// TwinCAT 3 PLC project TcoCore
// Title: TcoCore
// Company: Vortex.Library
// Author: Inxton
// ProjectVersion: 0.6.0.913
// ProgramVersion: 3.1.4024.12
// libraries:
//   Tc2_Standard, * (Beckhoff Automation GmbH)
//   Tc2_System, * (Beckhoff Automation GmbH)
//   Tc3_Module, * (Beckhoff Automation GmbH)
//   Tc2_EtherCAT,newest,Beckhoff Automation GmbH
//   Tc3_JsonXml,newest,Beckhoff Automation GmbH
// project tree:
//   / MAIN.TcPOU, PlcTask.TcTTO
//   POUs/Compatibility/ TcoContextCompatibility.TcPOU, TcoContextNfCompatibility.TcPOU
//   POUs/ImplicitChecks/ CheckBounds.TcPOU, CheckDivDInt.TcPOU, CheckDivLInt.TcPOU, CheckDivLReal.TcPOU, CheckDivReal.TcPOU, CheckLRangeSigned.TcPOU, CheckLRangeUnsigned.TcPOU, CheckPointer.TcPOU, CheckRangeSigned.TcPOU, CheckRangeUnsigned.TcPOU
//   POUs/Prototypes/Abstractions/ ITcoCoordinator.TcIO
//   POUs/Prototypes/TcoComponent/ ITcoComponent.TcIO, TcoComponent.TcPOU, TcoSignalInfo.TcPOU, ITcoServiceable.TcIO
//   POUs/Prototypes/TcoContext/ ITcoContextEnvironment.TcIO, TcoContextEnvironment.TcPOU, TcoContext.TcPOU, ITcoContext.TcIO
//   POUs/Prototypes/TcoDialog/TcoCustomizedDialog/ eCustomizedDialogAnswer.TcDUT, ITcoCustomizedDialogAnswer.TcIO (not stored), ITcoCustomizedDialogFormat.TcIO, TcoCustomizedDialog.TcPOU
//   POUs/Prototypes/TcoDialog/ eDialogAnswer.TcDUT, eDialogType.TcDUT, ITcoDialogAnswer.TcIO, ITcoDialogFormat.TcIO, TcoDialog.TcPOU, TcoDialogBase.TcPOU
//   POUs/Prototypes/TcoDialog/TcoInputDialog/ eInputDialogAnswer.TcDUT, ITcoInputDialogAnswer.TcIO, ITcoInputDialogFormat.TcIO, TcoInputDialog.TcPOU, TcoInputDialogContentContainer.TcPOU
//   POUs/Prototypes/TcoLogger/ ITcoLogger.TcIO, TcoLogger.TcPOU, TcoLogItem.TcDUT
//   POUs/Prototypes/TcoMessage/ eMessageCategory.TcDUT, eMessageCondition.TcDUT, eMessageDigestMethod.TcDUT, eMessengerLogMethod.TcDUT, ITcoMessageTextBuilder.TcIO, ITcoMessageProperties.TcIO, ITcoMessageCategorize.TcIO, ITcoMessenger.TcIO, ITcoMessengerEnv.TcIO, ITcoMessages.TcIO, TcoMessageDigest.TcDUT, TcoMessenger.TcPOU, TcoMessage.TcDUT, TcoMessengerEnv.TcPOU
//   POUs/Prototypes/TcoMomentaryTask/ ITcoMomentaryTask.TcIO, TcoMomentaryTask.TcPOU
//   POUs/Prototypes/TcoNothing/ NO.TcPOU
//   POUs/Prototypes/TcoObject/ ITcoObject.TcIO, TcoObject.TcPOU
//   POUs/Prototypes/TcoRemoteTask/ TcoRemoteTask.TcPOU
//   POUs/Prototypes/TcoRestorable/ ITcoObjectRestorer.TcIO, ITcoRestorable.TcIO
//   POUs/Prototypes/TcoRtc/ ITcoRtc.TcIO, RtcPrg.TcPOU, RtcSynchParams.TcDUT, TcoRtc.TcPOU
//   POUs/Prototypes/TcoSelector/ ITcoSelector.TcIO
//   POUs/Prototypes/TcoSequencer/ eStepIdUniquenessControlState.TcDUT, eSequencerMode.TcDUT, eStepStatus.TcDUT, eSequencerError.TcDUT, ITcoSequencerModeController.TcIO, TcoSequence.TcPOU, TcoSequencer.TcPOU, TcoSequencerModeController.TcPOU, TcoSequencerBase.TcPOU, ITcoSequencer.TcIO, StepDetails.TcDUT
//   POUs/Prototypes/TcoSequencer/TcoSequencerObserver/ ITcoSequencerObserver.TcIO, TcoSequencerObserver.TcPOU, TcoTcoSequencerObserverDummy.TcPOU
//   POUs/Prototypes/TcoState/ eRestoreMode.TcDUT, ITcoState.TcIO, TcoStateBase.TcPOU, TcoState.TcPOU, TcoStateExtendible.TcPOU
//   POUs/Prototypes/TcoStruct/ TcoParentedStructure.TcPOU, TcoStruct.TcDUT
//   POUs/Prototypes/TcoTask/ eTaskState.TcDUT, ITcoTaskStatus.TcIO, ITcoTask.TcIO, TcoTask.TcPOU
//   POUs/Prototypes/TcoTask/TaskResult/ TcoTaskResult.TcPOU, F_AnyToUnionValue.TcDUT
//   POUs/Prototypes/TcoTier/ TcoTier.TcPOU
//   POUs/Prototypes/TcoToggleTask/ ITcoToggleTask.TcIO, TcoToggleTask.TcPOU
//   POUs/TestFixtures/ _internals_TcoContext.TcPOU, _internals_TcoSequencer.TcPOU, _internals_TcoSequence.TcPOU
//   POUs/Utilities/ TcoCRC_16.TcPOU, TcoCRC_32.TcPOU, TcoCRC_8.TcPOU, StringBuilder.TcPOU
// real-time tasks:
//   TASK PlcTask: cycle T#10ms, priority 20, ADS port 350
//   TASK PlcTask1: cycle T#10ms, priority 21, ADS port 351
//   TASK PlcTask2: cycle T#10ms, priority 22, ADS port 352

CONFIGURATION TcoCore
    RESOURCE PLC ON TwinCAT3
        TASK PlcTask(INTERVAL := T#10ms, PRIORITY := 20);
        PROGRAM MAIN WITH PlcTask : MAIN;
    END_RESOURCE
END_CONFIGURATION

// ---- POUs/Prototypes/TcoDialog/TcoCustomizedDialog/eCustomizedDialogAnswer.TcDUT
{attribute 'qualified_only'}
{attribute 'strict'}
TYPE eCustomizedDialogAnswer :
(
    NoAnswer := 0,
    Option1 := 10,
    Option2 := 20,
    Option3 := 30,
    Option4 := 40,
    Invoked := 50
);
END_TYPE

// ---- POUs/Prototypes/TcoDialog/eDialogAnswer.TcDUT
{attribute 'qualified_only'}
{attribute 'strict'}
TYPE eDialogAnswer :
(
    NoAnswer := 0,
    OK := 10,
    Yes := 20,
    No := 30,
    Cancel := 40,
    Invoked := 50
);
END_TYPE

// ---- POUs/Prototypes/TcoDialog/eDialogType.TcDUT
{attribute 'qualified_only'}
{attribute 'strict'}
TYPE eDialogType :
(
    Undefined := 0,
    Info := 10,
    Question := 20,
    Warning := 30,
    Error := 40
);
END_TYPE

// ---- POUs/Prototypes/TcoDialog/TcoInputDialog/eInputDialogAnswer.TcDUT
{attribute 'qualified_only'}
{attribute 'strict'}
TYPE eInputDialogAnswer :
(
    NoAnswer := 0,
    OK := 10,
    Yes := 20,
    No := 30,
    Cancel := 40,
    Invoked := 50
);
END_TYPE

// ---- POUs/Prototypes/TcoLogger/TcoLogItem.TcDUT
(*~
    <docu>
        <summary>
            Logger message object contains complete message details including time stamp, message text, message category, identity of the message provider, context cycle in which the message was posted.
        </summary>
    </docu>
~*)
TYPE TcoLogItem :
STRUCT
    (*~
    <docu>
        <summary>
            Time when the message was posted.
        </summary>
    </docu>
~*)
    {attribute clr [ReadOnly()]}
    TimeStamp : DT;
    (*~
    <docu>
        <summary>
            Text of the message.
        </summary>
    </docu>
~*)
    {attribute clr [ReadOnly()]}
    Text : STRING(TcoMessengerEnv.MAX_MESSAGE_TEXT_LENGHT);
    (*~
    <docu>
        <summary>
            Identity of the TcoObject that posted this message.
        </summary>
    </docu>
~*)
    {attribute clr [ReadOnly()]}
    Identity : ULINT;
    (*~
    <docu>
        <summary>
            Message category of this message. See <see cref="TcoCore.eMessageCategory"/> for detailed informations.
        </summary>
    </docu>
~*)
    Category : eMessageCategory;
    (*~
    <docu>
        <summary>
            Context cycle in which the message was posted.
        </summary>
    </docu>
~*)
    {attribute clr [ReadOnly()]}
    Cycle : ULINT;
    (*~
    <docu>
        <summary>
            Count of messages of the object in the current cycle.
        </summary>
    </docu>
~*)
    {attribute clr [ReadOnly()]}
    PerCycleCount : BYTE;
    (*~
    <docu>
        <summary>
            Indicates that the message is expected to be dequeed from the buffer.
        </summary>
    </docu>
~*)
    ExpectDequeing : BOOL;
    (*~
    <docu>
        <summary>
            Stores message digest of this message text.
        </summary>
    </docu>
    ~*)
    MessageDigest : DWORD;
END_STRUCT
END_TYPE

// ---- POUs/Prototypes/TcoMessage/eMessageCategory.TcDUT
(*~
    <docu>
        <summary>
            Message categories.
        </summary>
    </docu>
~*)
// ATTENTION: Values must be multiply of 100
{attribute 'qualified_only'}
{attribute 'strict'}
TYPE eMessageCategory :
(
    All := 0,
    (*~
    <docu>
        <summary>
            Trace message to be used for tracing purpose.
            Use when you need to track detailed information about internal states of the program for detailed visibility.
            This is lowest level of category that can be used in production, for detailed observation of PLC program.
        </summary>
    </docu>
    ~*)
    Trace := 100,
    (*~
    <docu>
        <summary>
            Debug message to be used for debugging purpose only.
            Use when you need to report debug information for you as programmer.
        </summary>
    </docu>
    ~*)
    Debug := 200,
    (*~
    <docu>
        <summary>
            Info message.
            Use when you want to deliver information to the user, that has only informative character and does not adversely affect a process.
        </summary>
    </docu>
    ~*)
    Info := 300,
    (*~
    <docu>
        <summary>
            Time-out message.
            Use this category when you want to report a timed-out information, that may eventually succed.
        </summary>
    </docu>
    ~*)
    TimedOut := 400,
    (*~
    <docu>
        <summary>
            Notification message.
            Use this category when you want to report a notification that may be of interest to the user, but does not adversly affect a process.
        </summary>
    </docu>
    ~*)
    Notification := 500,
    (*~
    <docu>
        <summary>
            Warning message.
            Use this category when you want to report to the user an information about a possible problem, that may adversly affect a process.
            Information in this cateogory aims to help the user to identify a problem, the cause of such problem does not necessarily stops the process.
        </summary>
    </docu>
    ~*)
    Warning := 600,
    (*~
    <docu>
        <summary>
            Error message.
            Use this categoty when there is a failure that cannot be immediately recovered and an intervention is needed. This is typically a situation when a device fails
            to deliver expected result.
            Do not use this category to report information about failed process like measurement or detection.
        </summary>
    </docu>
    ~*)
    Error := 700,
    (*~
    <docu>
        <summary>
            Programming issue.
            Use this category to inform about a possible programming error, defect in settings or missing information at a level of programming or system or process settings.
        </summary>
    </docu>
    ~*)
    ProgrammingError := 900,
    (*~
    <docu>
        <summary>
            Critical error.
            Use this category when a critical error occured, that is not recoverable by the means of software (reset/restore) and but device still operates under such conditions; a detailed inspection and an expert action is required.
        </summary>
    </docu>
    ~*)
    Critical := 1000,
    (*~
    <docu>
        <summary>
            Fatal error.
            Use this category when a fatal error occured, that is not recoverable by the means of software (reset/restore) and a detailed inspection is required, the device is not able to continue without special intervention,
        </summary>
    </docu>
    ~*)
    Fatal := 1100,
    (*~
    <docu>
        <summary>
            Catastrophic error.
            Use this category when there is a situation when the device cannot continue operations due to irrecoverable failure.
        </summary>
    </docu>
    ~*)
    Catastrophic := 1200,
    None := 32000
);
END_TYPE

// ---- POUs/Prototypes/TcoMessage/eMessageCondition.TcDUT
{attribute 'qualified_only'}
{attribute 'strict'}
TYPE INTERNAL eMessageCondition :
(
    Unconditional := 0,
    Active := 10,
    Inactive := 20
);
END_TYPE

// ---- POUs/Prototypes/TcoMessage/eMessageDigestMethod.TcDUT
(*~
    <docu>
        <summary>
            Message digest methods used to create fingerprint of a message.
        </summary>
    </docu>
~*)
{attribute 'qualified_only'}
{attribute 'strict'}
TYPE eMessageDigestMethod :
(
    (*~
    <docu>
        <summary>
             Fastest method with highest probability of colisions.
        </summary>
    </docu>
    ~*)
    CRC8 := 8,
    (*~
    <docu>
        <summary>
             Moderate speed method with lower probability of colisions.
        </summary>
    </docu>
    ~*)
    CRC16 := 16,
    (*~
    <docu>
        <summary>
             Slowest speed method with relatively low probability of colisions.
        </summary>
    </docu>
    ~*)
    CRC32 := 32,
    (*~
    <docu>
        <summary>
             Messages are not digested the repeated messages won't be filtered out.
             Use this option on low performance devices.
        </summary>
    </docu>
    ~*)
    NONE := 32767
);
END_TYPE

// ---- POUs/Prototypes/TcoMessage/eMessengerLogMethod.TcDUT
(*~
    <docu>
        <summary>
            Message logging method. Determines how the messages will be pushed to the log buffer.
        </summary>
    </docu>
~*)
{attribute 'qualified_only'}
{attribute 'strict'}
TYPE eMessengerLogMethod :
(
    (*~
    <docu>
        <summary>
            Logs message when the occurence of the message content arises.
            If the message with the same content occurs in the n+1 cycle such message is not pushed.
        </summary>
    </docu>
    ~*)
    OnEventRisen := 100,
    (*~
    <docu>
        <summary>
            Logs message continuosly with not filtering.
            <note type="important">This method may easily overrun the circular message buffer.</note>
        </summary>
    </docu>
    ~*)
    Continuous := 200,
    (*~
    <docu>
        <summary>
            No logging.
        </summary>
    </docu>
    ~*)
    NoLogging := 300
);
END_TYPE

// ---- POUs/Prototypes/TcoMessage/TcoMessageDigest.TcDUT
TYPE TcoMessageDigest :
STRUCT
    Digest : DWORD;
    Cycle : ULINT;
    Count : ULINT;
    Category : eMessageCategory;
END_STRUCT
END_TYPE

// ---- POUs/Prototypes/TcoMessage/TcoMessage.TcDUT
(*~
    <docu>
        <summary>
            Complete message details including time stamp, message text, message category, identity of the message provider, context cycle in which the message was posted.
        </summary>
    </docu>
~*)
TYPE TcoMessage :
STRUCT
    (*~
    <docu>
        <summary>
            Time when the message was posted.
        </summary>
    </docu>
~*)
    {attribute clr [ReadOnly()]}
    TimeStamp : DT;
    (*~
    <docu>
        <summary>
            Text of the message.
        </summary>
    </docu>
~*)
    {attribute clr [ReadOnly()]}
    Text : STRING(TcoMessengerEnv.MAX_MESSAGE_TEXT_LENGHT);
    (*~
    <docu>
        <summary>
            Identity of the TcoObject that posted this message.
        </summary>
    </docu>
~*)
    {attribute clr [ReadOnly()]}
    Identity : ULINT;
    (*~
    <docu>
        <summary>
            Message category of this message. See <see cref="TcoCore.eMessageCategory"/> for detailed informations.
        </summary>
    </docu>
~*)
    Category : eMessageCategory;
    (*~
    <docu>
        <summary>
            Context cycle in which the message was posted.
        </summary>
    </docu>
~*)
    {attribute clr [ReadOnly()]}
    Cycle : ULINT;
    (*~
    <docu>
        <summary>
            Count of messages of the object in the current cycle.
        </summary>
    </docu>
~*)
    {attribute clr [ReadOnly()]}
    PerCycleCount : BYTE;
    (*~
    <docu>
        <summary>
            Indicates that the message is expected to be dequeed from the buffer.
        </summary>
    </docu>
~*)
    ExpectDequeing : BOOL;
    (*~
    <docu>
        <summary>
            Indicates that the message must be persisted in the alarm view until acknowledged.
        </summary>
    </docu>
    ~*)
    Pinned : BOOL;
    (*~
    <docu>
        <summary>
            Stores message digest of this message text.
        </summary>
    </docu>
    ~*)
    MessageDigest : DWORD;
END_STRUCT
END_TYPE

// ---- POUs/Prototypes/TcoRtc/RtcSynchParams.TcDUT
TYPE RtcSynchParams :
STRUCT
    synchContextIdentity : ULINT;
    doSynch : BOOL;
    syncAmsId : STRING;
    syncPeriod : UINT;
END_STRUCT
END_TYPE

// ---- POUs/Prototypes/TcoSequencer/eStepIdUniquenessControlState.TcDUT
{attribute 'qualified_only'}
{attribute 'strict'}
TYPE eStepIdUniquenessControlState :
(
    Deactivated := -1,
    NotYetStarted := 0,
    Requested := 10,
    Started := 20,
    Running := 40,
    Done := 200,
    Error := 255
);
END_TYPE

// ---- POUs/Prototypes/TcoSequencer/eSequencerMode.TcDUT
(*~
    <docu>
        <summary>
            Modes of the sequencer.
        </summary>
    </docu>
~*)
{attribute 'qualified_only'}
{attribute 'strict'}
TYPE eSequencerMode :
(
    (*~
    <docu>
        <summary>
            Invalid, no logic is executed.
        </summary>
    </docu>
~*)
    Invalid := -10,
    (*~
    <docu>
        <summary>
            Sequencer runs the steps of the sequence.
            (When cyclic mode is selected, next step is automatically started after the previous one has been completed.)
        </summary>
    </docu>
~*)
    CyclicMode := 0,
    (*~
    <docu>
        <summary>
            Sequencer is in mode of step-by-step operation. The current step completes the execution regularly.
            In this mode the Step Forward/Backward and manual step execution is available.
            <para>
                See <see cref="PlcDocu.TcoCore.TcoSequencerModeController.StepForward()"/> for detailed description.
                See <see cref="PlcDocu.TcoCore.TcoSequencerModeController.StepIn()"/> for detailed description.
                See <see cref="PlcDocu.TcoCore.TcoSequencerModeController.StepBackward()"/> for detailed description.
            </para>
        </summary>
    </docu>
~*)
    StepMode := 10
);
END_TYPE

// ---- POUs/Prototypes/TcoSequencer/eStepStatus.TcDUT
(*~
    <docu>
        <summary>
            Describes the step status inside the sequencer.
        </summary>
    </docu>
~*)
{attribute 'qualified_only'}
{attribute 'strict'}
TYPE eStepStatus :
(
    (*~
    <docu>
        <summary>
            No status defined.
        </summary>
    </docu>
~*)
    None := 0,
    (*~
    <docu>
        <summary>
            Step is disabled and won't be executed.
            Next enabled step in the sequence will be executed, when the sequencer reaches that step.
        </summary>
    </docu>
~*)
    Disabled := 10,
    (*~
    <docu>
        <summary>
            Step is ready to run. This case occurs when sequence is in step mode, step is in order of the execution and step is enabled.
            The body statements of the current step's are not executing. After calling StepIn method, step starts running the statements.
        </summary>
    </docu>
~*)
    ReadyToRun := 20,
    (*~
    <docu>
        <summary>
            Step is currently running (The body statements are running).
        </summary>
    </docu>
~*)
    Running := 30,
    (*~
    <docu>
        <summary>
            Step has finished (The body statements are not running).
        </summary>
    </docu>
~*)
    Done := 40,
    (*~
    <docu>
        <summary>
            Step is in error state. The sequencer does not execute any step logic.
        </summary>
    </docu>
~*)
    Error := 50
);
END_TYPE

// ---- POUs/Prototypes/TcoSequencer/eSequencerError.TcDUT
(*~
    <docu>
        <summary>
            Describes cause of the sequencer error.
        </summary>
    </docu>
~*)
{attribute 'qualified_only'}
{attribute 'strict'}
TYPE eSequencerError :
(
    (*~
    <docu>
        <summary>
            No error.
        </summary>
    </docu>
~*)
    noError := 0,
    (*~
    <docu>
        <summary>
            Some of the StepId in the sequence is not unique (```TcoSequencer.Step(StepID)```).
        </summary>
    </docu>
~*)
    NotUniqueStepId := 10,
    (*~
    <docu>
        <summary>
            StepId of the currently executed step has been changed during execution.
        </summary>
    </docu>
~*)
    StepIdHasBeenChanged := 20,
    (*~
    <docu>
        <summary>
            Order of the currently executed step has been changed during execution.
        </summary>
    </docu>
~*)
    OrderOfTheStepHasBeenChanged := 40,
    (*~
    <docu>
        <summary>
            Method ```RequestStep``` has been called with nonexisting StepId.
        </summary>
    </docu>
~*)
    StepWithRequestedIdDoesNotExists := 50,
    (*~
    <docu>
        <summary>
            Multiple simultaneous calls of ```RequestStep()```. Another ```RequestStep()``` method has been called while previous ```RequestStep()``` call has not yet been completed.
        </summary>
    </docu>
~*)
    MultipleRequestStepMethodCall := 60,
    (*~
    <docu>
        <summary>
            StepId is bellow min. range. Minimal value is -32767.
        </summary>
    </docu>
~*)
    StepIdTooLow := 70,
    (*~
    <docu>
        <summary>
            StepId is above max range. Maximal value is 32766.
        </summary>
    </docu>
~*)
    StepIdTooHigh := 80,
    (*~
    <docu>
        <summary>
            Mode of the sequencer is invalid.
        </summary>
    </docu>
~*)
    InvalidSequencerMode := 90
);
END_TYPE

// ---- POUs/Prototypes/TcoSequencer/StepDetails.TcDUT
(*~
    <docu>
        <summary>
            Describes the status of a step of the sequencer.
        </summary>
    </docu>
~*)
TYPE StepDetails :
STRUCT
    (*~
    <docu>
        <summary>
            Step identification number.
        </summary>
        <remarks>
             <note type="important">
                This number must be unique throughout the complete sequence. It is required to uniquely identify the step of the sequence.
            </note>
            <para>
                The <see cref="PlcDocu.TcoCore.TcoSequencer.RequestStep"/> method is using this number to jump to the required step.
            </para>
        </remarks>
    </docu>
~*)
    {attribute addProperty Name "<#Step ID#>"}
    ID : INT;
    (*~
    <docu>
        <summary>
            Order of the step in the sequence.
        </summary>
    </docu>
~*)
    {attribute addProperty Name "<#Step Order#>"}
    Order : UINT;
    (*~
    <docu>
        <summary>
            If this value is false, step body is not executed and execution is moved to the next enabled step in the sequence.
        </summary>
    </docu>
~*)
    {attribute addProperty Name "<#Enabled#>"}
    Enabled : BOOL;
    (*~
    <docu>
        <summary>
            Step description text.
        </summary>
    </docu>
~*)
    {attribute addProperty Name "<#Step description#>"}
    Description : STRING(254);
    (*~
    <docu>
        <summary>
            Describes step status.
        </summary>
        <remarks>
            <para>
                See <see cref="TcoCore.eStepStatus"/> for detailed description.
            </para>
        </remarks>
        enumStepStatus
    </docu>
~*)
    {attribute addProperty Name "<#Step status#>"}
    Status : eStepStatus;
    (*~
    <docu>
        <summary>
            Step duration time.
        </summary>
    </docu>
~*)
    {attribute addProperty Name "<#Step duration#>"}
    Duration : TIME;
END_STRUCT
END_TYPE

// ---- POUs/Prototypes/TcoState/eRestoreMode.TcDUT
{attribute 'qualified_only'}
{attribute 'strict'}
TYPE eRestoreMode :
(
    None := 0,
    (*~
    <docu>
        <summary>
                Activates automatic restore mechanism for all immediate children (direct members).
        </summary>
    </docu>
    ~*)
    AutoRestoreMembers := 10
);
END_TYPE

// ---- POUs/Prototypes/TcoStruct/TcoStruct.TcDUT
(*~
    <docu>
        <summary>
            Basic structure block from which most of the structures in TcOpen derive. `TcoStruct` provides construction mechanism to allow for access to the
            parent function block and the context.
            <note type="important">
                    The derived structure must be initialized in the declaration of the function block `mystruct : MyCustomStructure := (Parent := THIS^)`,
                    when nested in another structure `mystruct : MyCustomStructure := (Parent := THISSTRUCT)`. This will provide access to the `TcoContext`
                    and parent `TcoObject`.
            </note>
         </summary>

    </docu>
~*)
TYPE ABSTRACT TcoStruct :
STRUCT
    {attribute 'hide'}
    {attribute clr [ReadOnly()]}
    Parent : ITcoObject;
    (*~
        <docu>
            <summary>
                Provides access to parent object of this structure.
            </summary>
        </docu>
        ~*)
    {attribute 'hide'}
    {attribute clr [ReadOnly()]}
    {attribute clr [CompilerOmits("BuilderPlainer", "BuilderShadow")]}
    THISSTRUCT : TcoParentedStructure(NO.Obj, THIS^);
END_STRUCT
END_TYPE

// ---- POUs/Prototypes/TcoTask/eTaskState.TcDUT
(*~
    <docu>
        <summary>
            Describes the state of the respective task.
        </summary>
    </docu>
~*)
{attribute 'qualified_only'}
{attribute 'strict'}
TYPE eTaskState :
(
    (*~
    <docu>
        <summary>
            Task is in Ready state, the Execute() method returns FALSE.
            Task can be started by calling the Invoke() method.
        </summary>
    </docu>
~*)
    Ready := 0,
    (*~
    <docu>
        <summary>
            Task is in Requested state, if Invoke() method has been called and the Execute() method has not been called yet. The first following call of the method Execute()
            change the task state to Executing and returns TRUE, until Done or Error state is reached.
        </summary>
    </docu>
~*)
    Requested := 10,
    (*~
    <docu>
        <summary>
            When the task is in Busy state, Execute() method returns TRUE. Leaving this state is possible as follows:
            <para>1.) By calling the Abort() task gets into the Idle state.</para>
            <para>2.) By calling the DoneWhen(true) task gets into the Done state.</para>
            <para>3.) By calling the Restore() task gets into the Idle state.</para>
            <para>4.) By calling the ThrowWhen(true) task gets into the Error state.</para>
        </summary>
    </docu>
~*)
    Busy := 20,
    (*~
    <docu>
        <summary>
            Task is in Error state. To be able to start the task again the error state has to be reseted by calling the Restore() method.
        </summary>
    </docu>
~*)
    Error := 30,
    (*~
    <docu>
        <summary>
            Task is in Done state, Execute() method returns FALSE. To be able to start the task again '''rising edge''' of the calling of the Invoke() method needs to be performed.
            <p>Analogously to the xExecute signal of the <a href="https://plcopen.org/sites/default/files/downloads/creating_plcopen_compliant_function_block_libraries.pdf" title="Title"> PLCopen </a> motion function blocks.</p>
        </summary>
    </docu>
~*)
    Done := 40
);
END_TYPE

// ---- POUs/Prototypes/TcoTask/TaskResult/F_AnyToUnionValue.TcDUT
// credits Jakob Sagatowski https://github.com/sagatowski & contributors https://github.com/tcunit/TcUnit
TYPE F_AnyToUnionValue : UNION
    _bool : BOOL;
    _bit : BIT;
    _byte : BYTE;
    _dword : DWORD;
    _lword : LWORD;
    _string : STRING(255);
    _udint : UDINT;
    _uint : UINT;
    _usint : USINT;
    _sint : SINT;
    _int : INT;
    _word : WORD;
    _dint : DINT;
    _lint : LINT;
    _ulint : ULINT;
    _real : REAL;
    _lreal : LREAL;
    _wstring : WSTRING(255);
    _time : TIME;
    _ltime : LTIME;
    _date : DATE;
    _dateandtime : DATE_AND_TIME;
    _timeofday : TIME_OF_DAY;
END_UNION
END_TYPE

// ---- POUs/Prototypes/Abstractions/ITcoCoordinator.TcIO
INTERFACE ITcoCoordinator

PROPERTY IsFreshState : BOOL
GET
END_GET
END_PROPERTY

METHOD MoveNext : BOOL
END_METHOD

METHOD Retry : BOOL
VAR_INPUT
	inFromState : INT;
END_VAR
END_METHOD

METHOD Terminate : BOOL
END_METHOD

END_INTERFACE

// ---- POUs/Prototypes/TcoComponent/ITcoComponent.TcIO
INTERFACE ITcoComponent EXTENDS ITcoObject,ITcoRestorable, ITcoServiceable

END_INTERFACE

// ---- POUs/Prototypes/TcoContext/ITcoContextEnvironment.TcIO
INTERFACE ITcoContextEnvironment

PROPERTY Messaging : ITcoMessengerEnv
GET
END_GET
END_PROPERTY

END_INTERFACE

// ---- POUs/Prototypes/TcoDialog/TcoCustomizedDialog/ITcoCustomizedDialogFormat.TcIO
INTERFACE ITcoCustomizedDialogFormat

METHOD WithCaption : ITcoCustomizedDialogAnswer
VAR_INPUT
	inCaption : STRING(255);
END_VAR
END_METHOD

METHOD WithImage : ITcoCustomizedDialogAnswer
VAR_INPUT
	inSource : STRING(255);
	inHeight:REAL;
	inWidth:REAL;
END_VAR
END_METHOD

METHOD WithOption1 : ITcoCustomizedDialogAnswer
VAR_INPUT
	inContent:STRING;
END_VAR
END_METHOD

METHOD WithOption2 : ITcoCustomizedDialogAnswer
VAR_INPUT
	inContent:STRING;
END_VAR
END_METHOD

METHOD WithOption3 : ITcoCustomizedDialogAnswer
VAR_INPUT
	inContent:STRING;
END_VAR
END_METHOD

METHOD WithOption4 : ITcoCustomizedDialogAnswer
VAR_INPUT
	inContent:STRING;
END_VAR
END_METHOD

METHOD WithText : ITcoCustomizedDialogAnswer
VAR_INPUT
	inText : STRING(500);
END_VAR
END_METHOD

METHOD WithType : ITcoCustomizedDialogAnswer
VAR_INPUT
	inDialogType : eDialogType;
END_VAR
END_METHOD

END_INTERFACE

// ---- POUs/Prototypes/TcoDialog/ITcoDialogAnswer.TcIO
INTERFACE ITcoDialogAnswer EXTENDS ITcoDialogFormat

PROPERTY Answer : eDialogAnswer
GET
END_GET
END_PROPERTY

END_INTERFACE

// ---- POUs/Prototypes/TcoDialog/ITcoDialogFormat.TcIO
INTERFACE ITcoDialogFormat

METHOD WithCaption : ITcoDialogAnswer
VAR_INPUT
	inCaption : STRING(255);
END_VAR
END_METHOD

METHOD WithImage : ITcoDialogAnswer
VAR_INPUT
	inSource : STRING(255);
	inHeight:REAL;
	inWidth:REAL;
END_VAR
END_METHOD

METHOD WithOk : ITcoDialogAnswer
VAR_INPUT
END_VAR
END_METHOD

METHOD WithText : ITcoDialogAnswer
VAR_INPUT
	inText : STRING(500);
END_VAR
END_METHOD

METHOD WithType : ITcoDialogAnswer
VAR_INPUT
	inDialogType : eDialogType;
END_VAR
END_METHOD

METHOD WithYesNo : ITcoDialogAnswer
VAR_INPUT
END_VAR
END_METHOD

METHOD WithYesNoCancel : ITcoDialogAnswer
END_METHOD

END_INTERFACE

// ---- POUs/Prototypes/TcoDialog/TcoInputDialog/ITcoInputDialogAnswer.TcIO
INTERFACE ITcoInputDialogAnswer EXTENDS ITcoInputDialogFormat

PROPERTY Answer : eInputDialogAnswer
GET
END_GET
END_PROPERTY

END_INTERFACE

// ---- POUs/Prototypes/TcoDialog/TcoInputDialog/ITcoInputDialogFormat.TcIO
INTERFACE ITcoInputDialogFormat

METHOD WithCaption : ITcoInputDialogAnswer
VAR_INPUT
	inCaption : STRING(255);
END_VAR
END_METHOD

METHOD WithImage : ITcoInputDialogAnswer
VAR_INPUT
	inSource : STRING(255);
	inHeight:REAL;
	inWidth:REAL;
END_VAR
END_METHOD

METHOD WithOk : ITcoInputDialogAnswer
VAR_INPUT
END_VAR
END_METHOD

METHOD WithText : ITcoInputDialogAnswer
VAR_INPUT
	inText : STRING(500);
END_VAR
END_METHOD

METHOD WithType : ITcoInputDialogAnswer
VAR_INPUT
	inDialogType : eDialogType;
END_VAR
END_METHOD

METHOD WithYesNo : ITcoInputDialogAnswer
VAR_INPUT
END_VAR
END_METHOD

END_INTERFACE

// ---- POUs/Prototypes/TcoLogger/ITcoLogger.TcIO
INTERFACE ITcoLogger

(*~
		<docu>
			<summary>
				Pushes the message to logging buffer.
				See also `PushMessage`
				<note type="important">When using this method in a cyclical environment the message will be push each time it is called. You may easily overrun the logging buffer.</note>
			</summary>
		</docu>
~*)
METHOD PUBLIC Push
VAR_INPUT
	(*~
		<docu>
			<summary>
				Message/log entry text.
			</summary>
		</docu>
	~*)
	Text : STRING(TcoMessengerEnv.MAX_MESSAGE_TEXT_LENGHT);
	(*~
		<docu>
			<summary>
				Message/log entry category.
			</summary>
		</docu>
	~*)
	Category : eMessageCategory;
END_VAR
END_METHOD

(*~
		<docu>
			<summary>
				Pushes the message to logging buffer.
				See also `Push`
				<note:important>
						This method is typically invoked from a `TcoMessenger`.
						Depending on settings of the messenger the messages can be logged on rising edge of the message, to prevent buffer overrun.
						For details see `TcoMessengerSettings`.
				</note>
			</summary>
		</docu>
~*)
METHOD PushMessage
VAR_INPUT
	inMessage : TcoMessage;
END_VAR
END_METHOD

END_INTERFACE

// ---- POUs/Prototypes/TcoMessage/ITcoMessageTextBuilder.TcIO
INTERFACE ITcoMessageTextBuilder

METHOD Append : ITcoMessageTextBuilder
VAR_INPUT
	Text : STRING(TcoMessengerEnv.MAX_MESSAGE_TEXT_LENGHT);
END_VAR
END_METHOD

METHOD AppendAny : ITcoMessageTextBuilder
VAR_INPUT
	Data : ANY;
END_VAR
END_METHOD

METHOD As : ITcoMessageCategorize
END_METHOD

END_INTERFACE

// ---- POUs/Prototypes/TcoMessage/ITcoMessageProperties.TcIO
INTERFACE ITcoMessageProperties

METHOD Pin : ITcoMessageProperties
END_METHOD

PROPERTY Pinned : BOOL
GET
END_GET
END_PROPERTY

END_INTERFACE

// ---- POUs/Prototypes/TcoMessage/ITcoMessageCategorize.TcIO
INTERFACE ITcoMessageCategorize

(*~
		<docu>
			<summary>
				Categotizes and creates the message as 'debug'.
			</summary>
		</docu>
~*)
METHOD PUBLIC AsDebug : ITcoMessageProperties
END_METHOD

(*~
		<docu>
			<summary>
				Categotizes and creates the message as 'error'.
			</summary>
		</docu>
~*)
METHOD PUBLIC AsError : ITcoMessageProperties
END_METHOD

(*~
		<docu>
			<summary>
				Categotizes and creates the message as 'fatal'.
			</summary>
		</docu>
~*)
METHOD PUBLIC AsFatal : ITcoMessageProperties
END_METHOD

(*~
		<docu>
			<summary>
				Categotizes and creates the message as 'information'.
			</summary>
		</docu>
~*)
METHOD PUBLIC AsInfo : ITcoMessageProperties
END_METHOD

(*~
		<docu>
			<summary>
				Categotizes and creates the message as 'trace'.
			</summary>
		</docu>
~*)
METHOD PUBLIC AsTrace : ITcoMessageProperties
END_METHOD

(*~
		<docu>
			<summary>
				Categotizes and creates the message as 'warning'.
			</summary>
		</docu>
~*)
METHOD PUBLIC AsWarning : ITcoMessageProperties
END_METHOD

END_INTERFACE

// ---- POUs/Prototypes/TcoMessage/ITcoMessenger.TcIO
INTERFACE ITcoMessenger EXTENDS ITcoMessages

(*~
		<docu>
			<summary>
				Clears the message content.
				<remarks>
					<note type="important">
						This method is exposed for Rpc calls, for testing purposes. Rpc calls of this method must not be used in production code
					</note>
				</remarks>
			</summary>
		</docu>
~*)
METHOD Clear
END_METHOD

METHOD OnCondition : ITcoMessages
VAR_INPUT
	inCondition : BOOL;
END_VAR
END_METHOD

END_INTERFACE

// ---- POUs/Prototypes/TcoMessage/ITcoMessengerEnv.TcIO
INTERFACE ITcoMessengerEnv

PROPERTY IsSuspended : BOOL
GET
END_GET
END_PROPERTY

PROPERTY MessageDigestMethod : eMessageDigestMethod
GET
END_GET
SET
END_SET
END_PROPERTY

PROPERTY MessengerLoggingMethod : eMessengerLogMethod
GET
END_GET
SET
END_SET
END_PROPERTY

PROPERTY MinLevel : eMessageCategory
GET
END_GET
SET
END_SET
END_PROPERTY

METHOD Resume : BOOL
VAR_INPUT
END_VAR
END_METHOD

PROPERTY StringBuilder : REFERENCE TO StringBuilder
GET
END_GET
END_PROPERTY

METHOD Suspend
END_METHOD

END_INTERFACE

// ---- POUs/Prototypes/TcoMessage/ITcoMessages.TcIO
INTERFACE ITcoMessages

METHOD Build : ITcoMessageTextBuilder
END_METHOD

(*~
		<docu>
			<summary>
				Adds message of 'debug' category to the message queue.
			</summary>
		</docu>
~*)
METHOD PUBLIC Debug : ITcoMessageProperties
VAR_INPUT
	(*~
		<docu>
			<summary>
				Arbitrary message string.
			</summary>
		</docu>
	~*)
	Message : STRING(TcoMessengerEnv.MAX_MESSAGE_TEXT_LENGHT);
END_VAR
END_METHOD

(*~
		<docu>
			<summary>
				Adds message of 'error' category to the message queue.
			</summary>
		</docu>
~*)
METHOD PUBLIC Error : ITcoMessageProperties
VAR_INPUT
	(*~
		<docu>
			<summary>
				Arbitrary message string.
			</summary>
		</docu>
	~*)
	Message : STRING(TcoMessengerEnv.MAX_MESSAGE_TEXT_LENGHT);
END_VAR
END_METHOD

(*~
		<docu>
			<summary>
				Adds message of 'information' category to the message queue.
			</summary>
		</docu>
~*)
METHOD PUBLIC Info : ITcoMessageProperties
VAR_INPUT
	(*~
		<docu>
			<summary>
				Arbitrary message string.
			</summary>
		</docu>
	~*)
	Message : STRING(TcoMessengerEnv.MAX_MESSAGE_TEXT_LENGHT);
END_VAR
END_METHOD

(*~
		<docu>
			<summary>
				Adds message of 'notification' category to the message queue.
			</summary>
		</docu>
~*)
METHOD Notify  : ITcoMessageProperties
VAR_INPUT
	(*~
		<docu>
			<summary>
				Arbitrary message string.
			</summary>
		</docu>
	~*)
	Message : STRING(TcoMessengerEnv.MAX_MESSAGE_TEXT_LENGHT);
END_VAR
END_METHOD

(*~
		<docu>
			<summary>
				Adds message of given category to the message queue.
			</summary>
			<returns>Message index.</returns>
		</docu>
~*)
METHOD PUBLIC Post  : ITcoMessageProperties
VAR_INPUT
	(*~
		<docu>
			<summary>
				Arbitrary message string.
			</summary>
		</docu>
	~*)
	Message : STRING(TcoMessengerEnv.MAX_MESSAGE_TEXT_LENGHT);
	(*~
		<docu>
			<summary>
				Message category.
			</summary>
		</docu>
	~*)
	Category : eMessageCategory;
END_VAR
END_METHOD

(*~
		<docu>
			<summary>
				Adds message of 'programming error' category to the message queue.
			</summary>
		</docu>
~*)
METHOD PUBLIC Programming : ITcoMessageProperties
VAR_INPUT
	(*~
		<docu>
			<summary>
				Arbitrary message string.
			</summary>
		</docu>
	~*)
	Message : STRING(TcoMessengerEnv.MAX_MESSAGE_TEXT_LENGHT);
END_VAR
END_METHOD

(*~
		<docu>
			<summary>
				Adds message of 'trace' category to the message queue.
			</summary>
		</docu>
~*)
METHOD PUBLIC Trace : ITcoMessageProperties
VAR_INPUT
	(*~
		<docu>
			<summary>
				Arbitrary message string.
			</summary>
		</docu>
	~*)
	Message : STRING(TcoMessengerEnv.MAX_MESSAGE_TEXT_LENGHT);
END_VAR
END_METHOD

(*
	<docu>
		<summary>
			Unpins this messenger.
		</summary>
	</docu>
*)
METHOD UnPin
END_METHOD

(*~
		<docu>
			<summary>
				Adds message of 'warning' category to the message queue.
			</summary>
		</docu>
~*)
METHOD PUBLIC Warning : ITcoMessageProperties
VAR_INPUT
	(*~
		<docu>
			<summary>
				Arbitrary message string.
			</summary>
		</docu>
	~*)
	Message : STRING(TcoMessengerEnv.MAX_MESSAGE_TEXT_LENGHT);
END_VAR
END_METHOD

END_INTERFACE

// ---- POUs/Prototypes/TcoComponent/ITcoServiceable.TcIO
INTERFACE ITcoServiceable

PROPERTY IsService : BOOL
GET
END_GET
END_PROPERTY

METHOD PUBLIC Service
END_METHOD

END_INTERFACE

// ---- POUs/Prototypes/TcoContext/ITcoContext.TcIO
INTERFACE ITcoContext EXTENDS ITcoObject

PROPERTY EndCycleCount : ULINT
GET
END_GET
END_PROPERTY

PROPERTY Environment : ITcoContextEnvironment
GET
END_GET
END_PROPERTY

PROPERTY Logger : ITcoLogger
GET
END_GET
END_PROPERTY

PROPERTY RealTimeClock : ITcoRtc
GET
END_GET
END_PROPERTY

PROPERTY StartCycleCount : ULINT
GET
END_GET
END_PROPERTY

END_INTERFACE

// ---- POUs/Prototypes/TcoMomentaryTask/ITcoMomentaryTask.TcIO
INTERFACE ITcoMomentaryTask EXTENDS ITcoObject

(*~
	<docu>
		<summary>
			Use to set the state of the '''TcoMomentaryOnTask''' to the value '''FALSE'''.
		</summary>
	</docu>
~*)
METHOD Off : BOOL
END_METHOD

(*~
	<docu>
		<summary>
			Use to set the state of the '''TcoMomentaryOnTask''' to the value '''TRUE'''.
		</summary>
	</docu>
~*)
METHOD On : BOOL
END_METHOD

END_INTERFACE

// ---- POUs/Prototypes/TcoObject/ITcoObject.TcIO
INTERFACE ITcoObject EXTENDS __SYSTEM.IQueryInterface

{attribute 'hide'}
PROPERTY Context : ITcoContext
GET
END_GET
END_PROPERTY

PROPERTY Identity : ULINT
GET
END_GET
END_PROPERTY

END_INTERFACE

// ---- POUs/Prototypes/TcoRestorable/ITcoObjectRestorer.TcIO
INTERFACE ITcoObjectRestorer

(*~
	<docu>
		<summary>
			Ensures calling the <c>Restore()</c> method on the object entered.
			<para>
				<example>
				<note type="Example">
				<para>
					Possibility to use the fluent syntax.
				</para>
					<code>ChangeState(newState).RestoreObject(myFirstChildObject).RestoreObject(mySecondChildObject);</code>
				 </note>
				</example>
			</para>
		</summary>
	</docu>
~*)
METHOD RestoreObject : ITcoObjectRestorer
VAR_INPUT
	Obj : ITcoRestorable;
END_VAR
END_METHOD

END_INTERFACE

// ---- POUs/Prototypes/TcoRestorable/ITcoRestorable.TcIO
INTERFACE ITcoRestorable EXTENDS __SYSTEM.IQueryInterface

METHOD Restore : ITcoRestorable
END_METHOD

END_INTERFACE

// ---- POUs/Prototypes/TcoRtc/ITcoRtc.TcIO
INTERFACE ITcoRtc

PROPERTY IsSynchronized : BOOL
GET
END_GET
END_PROPERTY

PROPERTY IsValid : BOOL
GET
END_GET
END_PROPERTY

METHOD NowLocal : DATE_AND_TIME
END_METHOD

METHOD NowLocalAsTIMESTRUCT : Tc2_EtherCAT.Tc2_Utilities.TIMESTRUCT
END_METHOD

METHOD NowUTC : DATE_AND_TIME
END_METHOD

METHOD NowUTCAsTIMESTRUCT : Tc2_EtherCAT.Tc2_Utilities.TIMESTRUCT
END_METHOD

METHOD TickClock : ULINT
END_METHOD

END_INTERFACE

// ---- POUs/Prototypes/TcoSelector/ITcoSelector.TcIO
INTERFACE ITcoSelector EXTENDS ITcoState

METHOD RequestState
VAR_INPUT
	State : INT;
END_VAR
END_METHOD

END_INTERFACE

// ---- POUs/Prototypes/TcoSequencer/ITcoSequencerModeController.TcIO
INTERFACE ITcoSequencerModeController

(*~
	<docu>
		<summary>
			Gets or sets sequencer mode.
			<remarks>
				<para>
					See <see cref="TcoCore.eSequencerMode"/> for detailed description.
				</para>
			</remarks>
		</summary>
	</docu>
~*)
PROPERTY PUBLIC Mode : eSequencerMode
GET
END_GET
SET
END_SET
END_PROPERTY

(*~
	<docu>
		<summary>
			This method triggers StepBackward task, that decrements current step (variable: <c> TcoSequencer._theOrderOfTheCurrentlyExecutedStep</c> ), in case the sequencer is in step mode, and the current step is greather than zero.
		</summary>
	</docu>
~*)
METHOD PUBLIC FINAL StepBackward
END_METHOD

(*~
	<docu>
		<summary>
			This method triggers StepForward task, that increment current step (variable: <c>TcoSequencer._theOrderOfTheCurrentlyExecutedStep</c> ),
			in case the sequencer is in step mode, and the current step is lower than number of steps in th sequence (variable: <c>TcoSequencer._numberOfStepsInSequence</c> ).
		</summary>
	</docu>
~*)
METHOD PUBLIC FINAL StepForward
END_METHOD

(*~
	<docu>
		<summary>
			Triggers StepIn task, that changes the current step status from ReadyToRun to Running.
			This causes starting the execution of the body of the current step.
		</summary>
	</docu>
~*)
METHOD PUBLIC FINAL StepIn
END_METHOD

END_INTERFACE

// ---- POUs/Prototypes/TcoSequencer/TcoSequencerObserver/ITcoSequencerObserver.TcIO
INTERFACE ITcoSequencerObserver

METHOD Observe
VAR_INPUT

	(*~
	<docu>
		<summary>
			Indicates that a step is active.
		</summary>
	</docu>
	~*)

	inIsStepActive : BOOL;
	(*~
	<docu>
		<summary>
			Currently running step order.
		</summary>
	</docu>
	~*)

	inCurrentStepOrder : UINT;
	(*~
	<docu>
		<summary>
			Step identification number.
		</summary>
		<remarks>
 			<note type="important">
				This number must be unique throughout the complete sequence. It is required to uniquely identify the step of the sequence.
			</note>
			<para>
				The <see cref="PlcDocu.TcoCore.TcoSequencer.RequestStep"/> method is using this number to jump to the required step.
			</para>
		</remarks>
	</docu>
	~*)
		{attribute addProperty Name "<#Step ID#>"}
		inID: INT;
	(*~
		<docu>
			<summary>
				Order of the step in the sequence.
			</summary>
		</docu>
	~*)
		{attribute addProperty Name "<#Step Order#>"}
		inOrder: UINT;
	(*~
		<docu>
			<summary>
				If this value is false, step body is not executed and execution is moved to the next enabled step in the sequence.
			</summary>
		</docu>
	~*)
		{attribute addProperty Name "<#Enabled#>"}
		inEnabled: BOOL;
	(*~
		<docu>
			<summary>
				Step description text.
			</summary>
		</docu>
	~*)
		{attribute addProperty Name "<#Step description#>"}
		inDescription: STRING(254);
	(*~
		<docu>
			<summary>
				Describes step status.
			</summary>
			<remarks>
				<para>
					See <see cref="TcoCore.eStepStatus"/> for detailed description.
				</para>
			</remarks>
			enumStepStatus
		</docu>
	~*)
		{attribute addProperty Name "<#Step status#>"}
		inStatus : eStepStatus;
	(*~
		<docu>
			<summary>
				Step duration time.
			</summary>
		</docu>
	~*)
		{attribute addProperty Name "<#Step duration#>"}
		inDuration : TIME;

			(*~
		<docu>
			<summary>
				Total steps count;
			</summary>
		</docu>
	~*)
		{attribute addProperty Name "<#Step count#>"}
		inStepCount : UINT;
END_VAR
END_METHOD

END_INTERFACE

// ---- POUs/Prototypes/TcoSequencer/ITcoSequencer.TcIO
INTERFACE ITcoSequencer EXTENDS ITcoState

(*~
	<docu>
		<summary>
			Gets the information about the current step.
		</summary>
	</docu>
~*)
PROPERTY CurrentStep : REFERENCE TO StepDetails
GET
END_GET
END_PROPERTY

PROPERTY ModeController : ITcoSequencerModeController
GET
END_GET
END_PROPERTY

(*~
	<docu>
		<summary>
			<para>
				Ensures calling the Open(), Main() and Close() methods in the desired order.
				This method is final, so it cannot be overloaded. The InstanceName.Run() needs to be called cyclically inside the appropriate context.
			</para>
		</summary>
	</docu>
~*)
METHOD PUBLIC FINAL Run
END_METHOD

END_INTERFACE

// ---- POUs/Prototypes/TcoState/ITcoState.TcIO
INTERFACE ITcoState EXTENDS ITcoObject, ITcoRestorable

PROPERTY IsAutoRestoreEnabled : BOOL
GET
END_GET
END_PROPERTY

PROPERTY LastStateChangeCycle : ULINT
GET
END_GET
END_PROPERTY

METHOD RestoreObject : ITcoObjectRestorer
VAR_INPUT
	Obj : ITcoRestorable;
END_VAR
END_METHOD

PROPERTY State : INT
GET
END_GET
END_PROPERTY

END_INTERFACE

// ---- POUs/Prototypes/TcoTask/ITcoTaskStatus.TcIO
INTERFACE ITcoTaskStatus

PROPERTY Busy : BOOL
GET
END_GET
END_PROPERTY

PROPERTY Done : BOOL
GET
END_GET
END_PROPERTY

PROPERTY Error : BOOL
GET
END_GET
END_PROPERTY

END_INTERFACE

// ---- POUs/Prototypes/TcoTask/ITcoTask.TcIO
INTERFACE ITcoTask EXTENDS ITcoObject, ITcoRestorable

METHOD Abort
END_METHOD

PROPERTY Busy : BOOL
GET
END_GET
END_PROPERTY

PROPERTY Done : BOOL
GET
END_GET
END_PROPERTY

PROPERTY Error : BOOL
GET
END_GET
END_PROPERTY

(*~
	<docu>
		<summary>
			Use to start the execution of the task. The starting is possible from Ready state.
			<para>Moreover it is also possible to start the task again from Done state by performing the '''rising edge''' of the calling of the Invoke() method.</para>
			<p>Analogously to the xExecute signal of the <a href="https://plcopen.org/sites/default/files/downloads/creating_plcopen_compliant_function_block_libraries.pdf" title="Title"> PLCopen </a> motion function blocks.</p>
		</summary>
	</docu>
~*)
METHOD Invoke : ITcoTaskStatus
END_METHOD

END_INTERFACE

// ---- POUs/Prototypes/TcoToggleTask/ITcoToggleTask.TcIO
INTERFACE ITcoToggleTask EXTENDS ITcoObject

(*~
	<docu>
		<summary>
			Use to set the state of the '''TcoToggleTask''' to the value '''FALSE'''.
		</summary>
	</docu>
~*)
METHOD Off : BOOL
END_METHOD

(*~
	<docu>
		<summary>
			Use to set the state of the '''TcoToggleTask''' to the value '''TRUE'''.
		</summary>
	</docu>
~*)
METHOD On : BOOL
END_METHOD

(*~
	<docu>
		<summary>
			Use to toggle the state of the '''TcoToggleTask'''.
		</summary>
	</docu>
~*)
METHOD Toggle : BOOL
END_METHOD

END_INTERFACE

// ---- MAIN.TcPOU
PROGRAM INTERNAL MAIN
VAR
END_VAR

END_PROGRAM

// ---- POUs/Compatibility/TcoContextCompatibility.TcPOU
{attribute 'hide'}
{attribute clr [ExcludeFromApiDocumentation()]}
FUNCTION_BLOCK ABSTRACT TcoContextCompatibility EXTENDS TcoContext

{attribute 'hide'}
METHOD PROTECTED FINAL _Close
THIS^.Close();
END_METHOD

{attribute 'hide'}
METHOD PROTECTED FINAL _Open
THIS^.Open();
END_METHOD

END_FUNCTION_BLOCK

// ---- POUs/Prototypes/TcoContext/TcoContext.TcPOU
(*~
    <docu>
        <summary>
            Root construction container, provides context information for <c>TcoObjects</c> declared within its scope.
            This function block is ```abstract``` and cannot be instantiated.
            Use <see cref="PlcDocu.TcoCore.TcoContext.Run()"/> to run this context, ```Run``` method must be called only once per PLC Task cycle.
            Several 'TcoContext' instances can be declared and called inside one TwinCAT PlcTask, but only once per PLC cycle.
            The instance should not be accessed from several Twincat PlcTasks.
            Default implemenation of the 'TcoContext' allows its child members access properties <see cref="PlcDocu.TcoCore.TcoContext.StartCycleCount()"/>
            and <see cref="PlcDocu.TcoCore.TcoContext.EndCycleCount()"/>, messenger settings, rtc and other information related to the context of the running logic.
            <note type="tip">
                 A <c>TcoContext</c> can contain objects, components and PLC logic of one independent station of the machine,
                 while the another one can cover the same for another station.
            </note>
            <remarks>
                <note type="tip">
                    TwinCAT PlcTask and <see cref="PlcDocu.TcoCore.TcoTask()"/> refer to two different concepts.
                </note>
            </remarks>
        </summary>
        <example>
            Declaration part of the 'TcoContext' example.
        </example>
        <example>
                [!code-pas[Main](~/../TcOpen/src/TcoApplicationExamples/XaeAppExamples/PlcAppExamples/POUs/Context/VitoCorleone_Context.TcPOU?name=ContextExampleDeclarations)]
        </example>
        <example>
            Implementation part of the 'TcoContext' example.
        </example>
        <example>
                [!code-pas[Main](~/../TcOpen/src/TcoApplicationExamples/XaeAppExamples/PlcAppExamples/POUs/Context/VitoCorleone_Context.TcPOU?name=ContextExampleCode)]
        </example>
    </docu>
~*)
FUNCTION_BLOCK PUBLIC ABSTRACT TcoContext IMPLEMENTS ITcoContext
VAR
    (*~
        <docu>
            <summary>
                Identity of this <c>TcoContext</c>.
                This variable is used in the higher level applications,
                it allows to identify the context in SCADA like applications.
            </summary>
        </docu>
    ~*)
    {attribute clr [RenderIgnore()]}
    {attribute clr [ReadOnly()]}
    _Identity : ULINT;
    {attribute clr [ReadOnly()]}
    _startCycleCount : ULINT;
    {attribute clr [ReadOnly()]}
    _endCycleCount : ULINT;
    _messagingLevel : eMessageCategory;
    {attribute clr [ReadOnly()]}
    _rtc : TcoRtc;
    {attribute clr [RenderIgnore()]}
    _settings : TcoContextEnvironment;
    {attribute clr [RenderIgnore()]}
    _logger : TcoLogger(THIS^);
    _timeSychnMessenger : TcoMessenger(THIS^);
END_VAR

(*~
    <docu>
        <summary>
            This method is called implicitly at the entry point of this context (<see cref="PlcDocu.TcoCore.TcoContext.Run()"/>).
            <remarks>
                <note type="important">
                    Do not call this method explicitly!
                </note>
            </remarks>
        </summary>
    </docu>
~*)
METHOD INTERNAL FINAL Close
_endCycleCount := _startCycleCount;
END_METHOD

(*~
    <docu>
        <summary>
            Returns reference to this instance of the <see cref="PlcDocu.TcoCore.TcoContext()"/>.
        </summary>
    </docu>
~*)
PROPERTY Context : ITcoContext
GET
Context := THIS^;
END_GET
END_PROPERTY

(*~
    <docu>
        <summary>
            Gets the value of the counter incrememented by '1' at the end of each execution of this <see cref="PlcDocu.TcoCore.TcoContext()"/>.
        </summary>
    </docu>
~*)
PROPERTY EndCycleCount : ULINT
GET
EndCycleCount := _endCycleCount;
END_GET
END_PROPERTY

PROPERTY Environment : ITcoContextEnvironment
GET
Environment := _settings;
END_GET
END_PROPERTY

{attribute 'hide'}
METHOD FB_init : BOOL
VAR_INPUT
    bInitRetains : BOOL; // if TRUE, the retain variables are initialized (warm start / cold start)
    bInCopyCode : BOOL; // if TRUE, the instance afterwards gets moved into the copy code (online change)
END_VAR
_Identity := ADR(THIS^);
END_METHOD

(*~
    <docu>
        <summary>
            Returns the identity of this <see cref ="PlcDocu.TcoCore.TcoContext()"/>.
            This value is assigned when instantiated and cannot be changed at runtime.
            This member is used in the higher level applications.
        </summary>
    </docu>
~*)
PROPERTY Identity : ULINT
GET
Identity := _Identity;
END_GET
END_PROPERTY

(*~
        <docu>
            <summary>
                Gets logger for this context.
            </summary>
        </docu>
~*)
PROPERTY PUBLIC Logger : ITcoLogger
GET
Logger := _logger;
END_GET
END_PROPERTY

(*~
    <docu>
        <summary>
            Main method of the TcoContext. This is the entry point of any control logic that belongs to this context.
            The call of this method is ensured by calling the <c>InstanceName.Run()</c> method, and it must not be called explicitly.
            This method is abstract, and it must be overridden in derived block.
        </summary>
    </docu>
~*)
METHOD PROTECTED ABSTRACT Main
END_METHOD

(*~
    <docu>
        <summary>
            Called on entry into context. When overridden in derived class allows to execute an arbitrary logic prior to opening the context cycle.
            <remarks>
                <note type="important">
                    The method executes prior to opening the context. The context might not be properly initialized on first call.
                    Any information contained in the context at this point are from the last execution.
                </note>
            </remarks>
        </summary>
    </docu>
~*)
METHOD PROTECTED OnEntry
END_METHOD

(*~
    <docu>
        <summary>
            Called upon exit from the context. When overridden in derived class allows to execute an arbitrary logic after closing the context cycle.
        </summary>
    </docu>
~*)
METHOD PROTECTED OnExit
END_METHOD

(*~
    <docu>
        <summary>
            This method is called implicitly at the entry point of this context (<see cref="PlcDocu.TcoCore.TcoContext.Run()"/>).
            <remarks>
                <note type="important">
                    Do not call this method explicitly.
                </note>
            </remarks>
        </summary>
    </docu>
~*)
METHOD INTERNAL FINAL Open
_startCycleCount := _startCycleCount + 1;
_rtc.UpdateInternal();
END_METHOD

PROPERTY RealTimeClock : ITcoRtc
GET
RealTimeClock := _rtc;
END_GET
END_PROPERTY

(*~
    <docu>
        <summary>
            Syncronizes the Real Time Clock (RTC) from given source.
            <remarks>
                <note type="important">
                    There is single RTC source for entire application. All context share the same RTC source.
                </note>
            </remarks>
        </summary>
    </docu>
~*)
METHOD RtcSynchronize : REFERENCE TO TcoContext
VAR_INPUT
    (*~
        <docu>
            <summary>
                When called with true the synchronization mechanism executes.
            </summary>
        </docu>
    ~*)
    inDoSynch : BOOL;
    (*~
        <docu>
            <summary>
                ```AMS ID``` of the system against which RTC of this application will synchronize.
            </summary>
        </docu>
    ~*)
    inSyncAmsId : STRING;
    (*~
        <docu>
            <summary>
                Set the synchronisation period.
            </summary>
        </docu>
    ~*)
    inSyncPeriod : UINT;
END_VAR
VAR
    _RtcSynchParams : RtcSynchParams;
END_VAR
_RtcSynchParams.doSynch := inDoSynch;
_RtcSynchParams.syncAmsId := inSyncAmsId;
_RtcSynchParams.syncPeriod := inSyncPeriod;
_RtcSynchParams.synchContextIdentity := THIS^._Identity;
{warning disable C0357}
RtcPrg.Synchronize(_RtcSynchParams);
{warning enable C0357}
RtcSynchronize REF= THIS^;
_timeSychnMessenger.OnCondition(NOT THIS^.RealTimeClock.IsValid).Error('<#Real time clock is invalid!#>').Pin();

_timeSychnMessenger
    .OnCondition(THIS^.RealTimeClock.IsValid AND NOT THIS^.RealTimeClock.IsSynchronized).Warning('<#Real time clock is not sychronized.#>');
END_METHOD

(*~
    <docu>
        <summary>
            <para>
                This method executes of this context. It provided correct order of execution order of inner methods. Any logic of this context must be called within <see cref="PlcDocu.TcoCore.TcoContext.Main()"/>
                method. This method is final, so it cannot be overriden. The <c>InstanceName.Run()</c> needs to be called cyclically.
            </para>
        </summary>
    </docu>
~*)
METHOD PUBLIC FINAL Run
THIS^.OnEntry();
THIS^.Open();
THIS^.Main();
THIS^.Close();
THIS^.OnExit();
END_METHOD

(*~
    <docu>
        <summary>
            Gets number of executions of this context. Value of this property is incremented by '1' at the beginning of the <see cref="PlcDocu.TcoCore.TcoContext()"/>.
        </summary>
    </docu>
~*)
PROPERTY StartCycleCount : ULINT
GET
StartCycleCount := _startCycleCount;
END_GET
END_PROPERTY

END_FUNCTION_BLOCK

// ---- POUs/Prototypes/TcoRtc/TcoRtc.TcPOU
FUNCTION_BLOCK PUBLIC TcoRtc IMPLEMENTS ITcoRtc
VAR
    {attribute 'hide'}
    _isValid : BOOL := FALSE;
    {attribute 'hide'}
    _state : UINT;
    {attribute 'hide'}
    _TimeZoneID : Tc2_EtherCAT.Tc2_Utilities.E_TimeZoneID;
    {attribute 'hide'}
    _NT_GetLocalTime : Tc2_EtherCAT.Tc2_Utilities.NT_GetTime;
    {attribute 'hide'}
    _FB_TzSpecificLocalTimeToSystemTime : Tc2_EtherCAT.Tc2_Utilities.FB_TzSpecificLocalTimeToSystemTime;
    {attribute 'hide'}
    _RTC_EX2 : Tc2_EtherCAT.Tc2_Utilities.RTC_EX2;
    {attribute 'hide'}
    _PDT : Tc2_EtherCAT.Tc2_Utilities.TIMESTRUCT;
    {attribute 'hide'}
    _LocalTime : Tc2_EtherCAT.Tc2_Utilities.TIMESTRUCT;
    {attribute clr [ReadOnly()]}
    _LocalTimeDT : DATE_AND_TIME;
    {attribute 'hide'}
    _UTCTime : Tc2_EtherCAT.Tc2_Utilities.TIMESTRUCT;
    {attribute clr [ReadOnly()]}
    _UTCTimeDT : DATE_AND_TIME;
END_VAR

PROPERTY IsSynchronized : BOOL
GET
IsSynchronized := RtcPrg._isSynchronized;
END_GET
END_PROPERTY

PROPERTY IsValid : BOOL
GET
IsValid := _isValid;
END_GET
END_PROPERTY

METHOD NowLocal : DATE_AND_TIME
IF _isValid THEN
    NowLocal := _LocalTimeDT;
END_IF
END_METHOD

METHOD NowLocalAsTIMESTRUCT : Tc2_EtherCAT.Tc2_Utilities.TIMESTRUCT
IF _isValid THEN
    NowLocalAsTIMESTRUCT := _LocalTime;
END_IF
END_METHOD

METHOD NowUTC : DATE_AND_TIME
IF _isValid THEN
    NowUTC := _UTCTimeDT;
END_IF
END_METHOD

METHOD NowUTCAsTIMESTRUCT : Tc2_EtherCAT.Tc2_Utilities.TIMESTRUCT
IF _isValid THEN
    NowUTCAsTIMESTRUCT := _UTCTime;
END_IF
END_METHOD

METHOD TickClock : ULINT
TickClock := Tc2_EtherCAT.F_GetActualDcTime64();
END_METHOD

METHOD PROTECTED Update
VAR
    _diffToLastSyncInSeconds : LINT;
END_VAR
IF _state = 0 THEN
    //	_isValid := FALSE;
    _NT_GetLocalTime(NETID := '127.0.0.1.1.1', START := TRUE);

    IF _NT_GetLocalTime.BUSY AND NOT _NT_GetLocalTime.ERR THEN
        _state := _state + 10;
    END_IF
END_IF

IF _state = 10 THEN
    _NT_GetLocalTime(START := FALSE);

    IF NOT _NT_GetLocalTime.BUSY AND NOT _NT_GetLocalTime.ERR THEN
        _state := _state + 10;
    END_IF
END_IF

IF _state = 20 THEN
    _NT_GetLocalTime(START := FALSE);
    _PDT := _NT_GetLocalTime.TIMESTR;
    _isValid := TRUE;
END_IF

_RTC_EX2(EN := _isValid, PDT := _PDT);

_diffToLastSyncInSeconds := ABS(ULINT_TO_LINT(Tc2_EtherCAT.SYSTEMTIME_TO_DCTIME64(_RTC_EX2.CDT, 0, 0) -
            Tc2_EtherCAT.SYSTEMTIME_TO_DCTIME64(RtcPrg._LastSyncTimeStampInLocalTime, 0, 0))) /
    1000000000;

IF _state >= 20 AND RtcPrg._RtcSynchParams.doSynch AND _diffToLastSyncInSeconds >= RtcPrg._RtcSynchParams.syncPeriod THEN
    _state := 0;
END_IF

_LocalTime := _RTC_EX2.CDT;
_LocalTimeDT := Tc2_EtherCAT.Tc2_Utilities.SYSTEMTIME_TO_DT(_LocalTime);

IF RtcPrg._isSynchronized THEN
    _FB_TzSpecificLocalTimeToSystemTime(in := _LocalTime,
        tzInfo := RtcPrg._TimeZoneInformation,
        out => _UTCTime,
        eTzID => _TimeZoneID);

    _UTCTimeDT := Tc2_EtherCAT.Tc2_Utilities.SYSTEMTIME_TO_DT(_UTCTime);
END_IF
END_METHOD

METHOD INTERNAL UpdateInternal
THIS^.Update();
END_METHOD

END_FUNCTION_BLOCK

// ---- POUs/Prototypes/TcoRtc/RtcPrg.TcPOU
{attribute 'obsolete' := 'Should not be accessed from outside TcoCore library. Publicly accesible due to compatibility reasons.'}
PROGRAM PUBLIC RtcPrg
VAR
    {attribute 'hide'}
    _RtcSynchParams : RtcSynchParams;
    {attribute 'hide'}
    _isSynchronized : BOOL := FALSE;
    {attribute 'hide'}
    _state : UINT;
    {attribute 'hide'}
    _syncAmsIdIsLocale : BOOL;
    {attribute 'hide'}
    _FB_GetLocalAmsNetId : Tc2_EtherCAT.Tc2_Utilities.FB_GetLocalAmsNetId;
    {attribute 'hide'}
    _FB_GetTimeZoneInformation : Tc2_EtherCAT.Tc2_Utilities.FB_GetTimeZoneInformation;
    {attribute 'hide'}
    _FB_SetTimeZoneInformation : Tc2_EtherCAT.Tc2_Utilities.FB_SetTimeZoneInformation;
    {attribute 'hide'}
    _TimeZoneInformation : Tc2_EtherCAT.Tc2_Utilities.ST_TimeZoneInformation;
    {attribute 'hide'}
    _TimeZoneID : Tc2_EtherCAT.Tc2_Utilities.E_TimeZoneID;
    {attribute 'hide'}
    _startTime : Tc2_EtherCAT.T_DCTIME64;
    {attribute 'hide'}
    _endTime : Tc2_EtherCAT.T_DCTIME64;
    {attribute 'hide'}
    _getOffset : Tc2_EtherCAT.T_DCTIME64;
    {attribute 'hide'}
    _setOffset : Tc2_EtherCAT.T_DCTIME64;
    {attribute 'hide'}
    _NT_GetSyncTime : Tc2_EtherCAT.Tc2_Utilities.NT_GetTime;
    {attribute 'hide'}
    _NT_SetLocalTime : Tc2_EtherCAT.Tc2_Utilities.NT_SetLocalTime;
    {attribute 'hide'}
    _NT_GetLocalTime : Tc2_EtherCAT.Tc2_Utilities.NT_GetTime;
    {attribute 'hide'}
    _FB_TzSpecificLocalTimeToSystemTime : Tc2_EtherCAT.Tc2_Utilities.FB_TzSpecificLocalTimeToSystemTime;
    {attribute 'hide'}
    _remote2localDiff : Tc2_EtherCAT.T_DCTIME64;
    {attribute 'hide'}
    _local2SyncDiff_nanoseconds : LINT;
    {attribute 'hide'}
    _offset : ULINT;
    {attribute 'hide'}
    _syncCounter : ULINT;
    {attribute 'hide'}
    _lastSyncTick : Tc2_EtherCAT.T_DCTIME64;
    {attribute 'hide'}
    _timeTick : Tc2_EtherCAT.T_DCTIME64;
    {attribute 'hide'}
    _LocalTime : Tc2_EtherCAT.Tc2_Utilities.TIMESTRUCT;
    {attribute 'hide'}
    _UTCTime : Tc2_EtherCAT.Tc2_Utilities.TIMESTRUCT;
    {attribute 'hide'}
    _syncStartLocalTime : Tc2_EtherCAT.Tc2_Utilities.TIMESTRUCT;
    {attribute 'hide'}
    _LastSyncTimeStampInLocalTime : Tc2_EtherCAT.Tc2_Utilities.TIMESTRUCT;
    {attribute 'hide'}
    _LastSyncDiff_seconds : LINT;
END_VAR

{attribute 'obsolete' := 'MUST NOT BE CALLED EXPLICITELY!!! Use TcoCore.TcoContext.RtcSynchronize() instead!!!'}
METHOD PUBLIC Synchronize
VAR_INPUT
    inRtcSynchParams : RtcSynchParams;
END_VAR
//If there is no synchronization context identity already set, the value of this identity is used.
//So first TcoContext that calls this method set the synchronization parameters.
IF _RtcSynchParams.synchContextIdentity = 0 AND inRtcSynchParams.synchContextIdentity <> 0 THEN
    _RtcSynchParams.synchContextIdentity := inRtcSynchParams.synchContextIdentity;
END_IF

//In case that another TcoContest calls this method, it is ignored as only one could set the synchronization parameters.
IF _RtcSynchParams.synchContextIdentity <> 0 AND _RtcSynchParams.synchContextIdentity = inRtcSynchParams.synchContextIdentity THEN
    _RtcSynchParams.doSynch := inRtcSynchParams.doSynch;
    _RtcSynchParams.syncAmsId := inRtcSynchParams.syncAmsId;
    _RtcSynchParams.syncPeriod := inRtcSynchParams.syncPeriod;

    IF _NT_GetLocalTime.ERR THEN
        _NT_GetLocalTime(START := FALSE);
        _isSynchronized := FALSE;
        RETURN;
    END_IF

    IF _state = 0 THEN
        IF _RtcSynchParams.doSynch THEN
            _isSynchronized := FALSE;
            _state := _state + 10;
        ELSE
            _isSynchronized := FALSE;
            _state := 210;
        END_IF
    END_IF

    IF _state = 10 THEN
        _syncStartLocalTime := _NT_GetLocalTime.TIMESTR;
        _FB_GetLocalAmsNetId(bExecute := TRUE);

        IF _FB_GetLocalAmsNetId.bBusy AND NOT _FB_GetLocalAmsNetId.bError THEN
            _state := _state + 10;
        END_IF
    END_IF

    IF _state = 20 THEN
        _FB_GetLocalAmsNetId(bExecute := FALSE);

        IF NOT _FB_GetLocalAmsNetId.bBusy AND NOT _FB_GetLocalAmsNetId.bError THEN
            _state := _state + 10;
        END_IF
    END_IF

    IF _state = 30 THEN
        _syncAmsIdIsLocale := _RtcSynchParams.syncAmsId = _FB_GetLocalAmsNetId.AddrString OR
            _RtcSynchParams.syncAmsId = '127.0.0.1.1.1' OR
            _RtcSynchParams.syncAmsId = '';

        _state := _state + 10;
    END_IF

    IF _state = 40 THEN
        _startTime := Tc2_EtherCAT.F_GetActualDcTime64();
        _state := _state + 10;
    END_IF

    IF _state = 50 THEN
        _FB_GetTimeZoneInformation(sNetID := _RtcSynchParams.syncAmsId, bExecute := TRUE);

        IF _FB_GetTimeZoneInformation.bBusy AND NOT _FB_GetTimeZoneInformation.bError THEN
            _state := _state + 10;
        END_IF
    END_IF

    IF _state = 60 THEN
        _FB_GetTimeZoneInformation(bExecute := FALSE);

        IF NOT _FB_GetTimeZoneInformation.bBusy AND NOT _FB_GetTimeZoneInformation.bError THEN
            _state := _state + 10;
        END_IF
    END_IF

    IF _state = 70 THEN
        _TimeZoneInformation := _FB_GetTimeZoneInformation.tzInfo;
        _TimeZoneID := _FB_GetTimeZoneInformation.tzID;
        _endTime := Tc2_EtherCAT.F_GetActualDcTime64();
        _getOffset := (_endTime - _startTime) / 2;
        _state := _state + 10;
    END_IF

    IF _state = 80 THEN
        IF _syncAmsIdIsLocale THEN
            _state := 180;
        ELSE
            _state := _state + 10;
        END_IF
    END_IF

    IF _state = 90 THEN
        _startTime := Tc2_EtherCAT.F_GetActualDcTime64();
        _state := _state + 10;
    END_IF

    IF _state = 100 THEN
        _FB_SetTimeZoneInformation(sNetID := '127.0.0.1.1.1', tzInfo := _TimeZoneInformation, bExecute := TRUE);

        IF _FB_SetTimeZoneInformation.bBusy AND NOT _FB_SetTimeZoneInformation.bError THEN
            _state := _state + 10;
        END_IF
    END_IF

    IF _state = 110 THEN
        _FB_SetTimeZoneInformation(bExecute := FALSE);

        IF NOT _FB_SetTimeZoneInformation.bBusy AND NOT _FB_SetTimeZoneInformation.bError THEN
            _state := _state + 10;
        END_IF
    END_IF

    IF _state = 120 THEN
        _endTime := Tc2_EtherCAT.F_GetActualDcTime64();
        _setOffset := (_endTime - _startTime) / 2;
        _state := _state + 10;
    END_IF

    IF _state = 130 THEN
        _NT_GetSyncTime(NETID := _RtcSynchParams.syncAmsId, START := TRUE);

        IF _NT_GetSyncTime.BUSY AND NOT _NT_GetSyncTime.ERR THEN
            _state := _state + 10;
        END_IF
    END_IF

    IF _state = 140 THEN
        _NT_GetSyncTime(START := FALSE);

        IF NOT _NT_GetSyncTime.BUSY AND NOT _NT_GetSyncTime.ERR THEN
            _state := _state + 10;
        END_IF
    END_IF

    IF _state = 150 THEN
        _NT_GetSyncTime(START := FALSE);
        _offset := LREAL_TO_ULINT(ULINT_TO_LREAL(_getOffset + _setOffset) / 1000000) * 1000000;
        _offset := _offset + Tc2_EtherCAT.SYSTEMTIME_TO_DCTIME64(_NT_GetSyncTime.TIMESTR, 0, 0) + _getOffset + _setOffset;
        _LocalTime := Tc2_EtherCAT.DCTIME64_TO_SYSTEMTIME(_offset);
        _state := _state + 10;
    END_IF

    IF _state = 160 THEN
        _NT_GetSyncTime(START := FALSE);
        _NT_SetLocalTime(NETID := '127.0.0.1.1.1', TIMESTR := _LocalTime, START := TRUE);

        IF _NT_SetLocalTime.BUSY AND NOT _NT_SetLocalTime.ERR THEN
            _state := _state + 10;
        END_IF
    END_IF

    IF _state = 170 THEN
        _NT_GetSyncTime(START := FALSE);
        _NT_SetLocalTime(START := FALSE);

        IF NOT _NT_SetLocalTime.BUSY AND NOT _NT_SetLocalTime.ERR THEN
            _state := _state + 10;
        END_IF
    END_IF

    IF _state = 180 THEN
        _NT_GetSyncTime(NETID := _RtcSynchParams.syncAmsId, START := TRUE);
        _NT_GetLocalTime(NETID := '127.0.0.1.1.1', START := TRUE);

        IF _NT_GetSyncTime.BUSY AND NOT _NT_GetSyncTime.ERR AND NOT _NT_GetLocalTime.ERR THEN
            _state := _state + 10;
        END_IF
    END_IF

    IF _state = 190 THEN
        _NT_GetSyncTime(START := FALSE);
        _NT_GetLocalTime(START := FALSE);

        IF NOT _NT_GetSyncTime.BUSY AND NOT _NT_GetSyncTime.ERR AND NOT _NT_GetLocalTime.BUSY AND NOT _NT_GetLocalTime.ERR THEN
            _state := _state + 10;
        END_IF
    END_IF

    IF _state = 200 THEN
        _LastSyncTimeStampInLocalTime := _NT_GetLocalTime.TIMESTR;

        _LastSyncDiff_seconds := ULINT_TO_LINT(Tc2_EtherCAT.SYSTEMTIME_TO_DCTIME64(_LastSyncTimeStampInLocalTime, 0, 0) -
                Tc2_EtherCAT.SYSTEMTIME_TO_DCTIME64(_syncStartLocalTime, 0, 0)) /
            1000000000;

        _local2SyncDiff_nanoseconds := ULINT_TO_LINT(Tc2_EtherCAT.SYSTEMTIME_TO_DCTIME64(_NT_GetLocalTime.TIMESTR, 0, 0) -
                Tc2_EtherCAT.SYSTEMTIME_TO_DCTIME64(_NT_GetSyncTime.TIMESTR, 0, 0));

        _NT_GetSyncTime(START := FALSE);
        _NT_GetLocalTime(START := FALSE);
        _NT_SetLocalTime(START := FALSE);
        _LocalTime := _NT_GetLocalTime.TIMESTR;

        _FB_TzSpecificLocalTimeToSystemTime(in := _LocalTime,
            tzInfo := _TimeZoneInformation,
            out => _UTCTime,
            eTzID => _TimeZoneID);

        _lastSyncTick := Tc2_EtherCAT.F_GetActualDcTime64();
        _syncCounter := _syncCounter + 1;
        _state := _state + 10;
    END_IF

    IF _state = 210 THEN
        _NT_GetLocalTime(NETID := '127.0.0.1.1.1', START := TRUE);

        IF _NT_GetLocalTime.BUSY AND NOT _NT_GetLocalTime.ERR THEN
            _state := _state + 10;
        END_IF
    END_IF

    IF _state = 220 THEN
        _NT_GetLocalTime(START := FALSE);

        IF NOT _NT_GetLocalTime.BUSY AND NOT _NT_GetLocalTime.ERR THEN
            _state := _state + 10;
        END_IF
    END_IF

    IF _state = 230 THEN
        _isSynchronized := TRUE;
        _NT_GetSyncTime(START := FALSE);
        _NT_GetLocalTime(START := FALSE);
        _NT_SetLocalTime(START := FALSE);
        _timeTick := Tc2_EtherCAT.F_GetActualDcTime64();

        IF _RtcSynchParams.doSynch THEN
            IF (_timeTick - _lastSyncTick) / 1000000000 >= _RtcSynchParams.syncPeriod THEN //Ticks are in nanoseconds, sync period is in seconds
                _state := 0;
            ELSE
                _state := 210;
            END_IF
        ELSE
            _state := 210;
        END_IF
    END_IF
END_IF
END_METHOD

END_PROGRAM

// ---- POUs/Prototypes/TcoContext/TcoContextEnvironment.TcPOU
FUNCTION_BLOCK TcoContextEnvironment IMPLEMENTS ITcoContextEnvironment
VAR
    {attribute clr [RenderIgnore()]}
    _messenger : TcoMessengerEnv;
END_VAR

(*~
        <docu>
            <summary>
                Gets messaging settings of this context.
            </summary>
        </docu>
~*)
PROPERTY Messaging : ITcoMessengerEnv
GET
Messaging := _messenger;
END_GET
END_PROPERTY

END_FUNCTION_BLOCK

// ---- POUs/Prototypes/TcoMessage/TcoMessengerEnv.TcPOU
FUNCTION_BLOCK PUBLIC TcoMessengerEnv IMPLEMENTS ITcoMessengerEnv
VAR
    _minLevel : eMessageCategory;
    _isMessagingSuspended : BOOL;
    _messageDigestMethod : eMessageDigestMethod := eMessageDigestMethod.CRC16;
    _messengerLoggingMethod : eMessengerLogMethod := eMessengerLogMethod.OnEventRisen;
    {attribute 'hide'}
    _sb : StringBuilder();
END_VAR
VAR CONSTANT
    MAX_MESSAGE_TEXT_LENGHT : INT := 160;
END_VAR

(*~
    <docu>
        <summary>
            Gets whether the messaging is suspended at this point in program.
            <para>
                See also <see cref="PlcDocu.TcoCore.TcoMessengerSettings.Resume()"/>
            </para>
            <para>
                See also <see cref="PlcDocu.TcoCore.TcoMessengerSettings.Suspend()"/>
            </para>
            <para>
                See also <see cref="PlcDocu.TcoCore.TcoMessengerSettings.MinLevel"/>
            </para>
        </summary>
    </docu>
~*)
PROPERTY PUBLIC IsSuspended : BOOL
GET
IsSuspended := _isMessagingSuspended;
END_GET
END_PROPERTY

(*~
    <docu>
        <summary>
            Gets or sets message digest method.
            Message digest serves to fingerprint messages.
            See also MessengerLoggingMethod.
        </summary>
    </docu>
~*)
PROPERTY MessageDigestMethod : eMessageDigestMethod
GET
MessageDigestMethod := _messageDigestMethod;
END_GET
SET
_messageDigestMethod := MessageDigestMethod;
END_SET
END_PROPERTY

(*~
    <docu>
        <summary>
            Gets or sets logging method.
            Logger can ingest messages continuously, on rising edge of a message or disable the logging.
        </summary>
    </docu>
~*)
PROPERTY MessengerLoggingMethod : eMessengerLogMethod
GET
MessengerLoggingMethod := _messengerLoggingMethod;
END_GET
SET
_messengerLoggingMethod := MessengerLoggingMethod;
END_SET
END_PROPERTY

(*~
    <docu>
        <summary>
            Gets or set minimal messaging level, the objects will post only messages for the levels of this or superior severity.
            <para>
                See also <see cref="PlcDocu.TcoCore.TcoMessengerSettings.Resume()"/>
            </para>
            <para>
                See also <see cref="PlcDocu.TcoCore.TcoMessengerSettings.Suspend()"/>
            </para>
            <para>
                See also <see cref="PlcDocu.TcoCore.TcoMessengerSettings.MinLevel"/>
            </para>
        </summary>
    </docu>
~*)
PROPERTY PUBLIC MinLevel : eMessageCategory
GET
MinLevel := _minLevel;
END_GET
SET
_minLevel := MinLevel;
END_SET
END_PROPERTY

(*~
    <docu>
        <summary>
            Resumes messaging from the all objects of this context, when the messaging was previously suspended by ```Suspend``` method.
            <para>
                See also <see cref="PlcDocu.TcoCore.TcoMessengerSettings.Suspend()"/>
            </para>
            <para>
                See also <see cref="PlcDocu.TcoCore.TcoMessengerSettings.MinLevel"/>
            </para>
        </summary>
    </docu>
~*)
METHOD PUBLIC Resume : BOOL
_isMessagingSuspended := FALSE;
END_METHOD

PROPERTY StringBuilder : REFERENCE TO StringBuilder
GET
StringBuilder REF= _sb;
END_GET
END_PROPERTY

(*~
    <docu>
        <summary>
            Suspends messaging from the all objects of this context that would occur from this point in the call tree.
            <para>
                See also <see cref="PlcDocu.TcoCore.TcoMessengerSettings.Resume()"/>
            </para>
            <para>
                See also <see cref="PlcDocu.TcoCore.TcoMessengerSettings.MinLevel"/>
            </para>
        </summary>
    </docu>
~*)
METHOD PUBLIC Suspend
_isMessagingSuspended := TRUE;
END_METHOD

END_FUNCTION_BLOCK

// ---- POUs/Utilities/StringBuilder.TcPOU
(*~
<docu>
    <summary>
            Allows to concat strings using fluent interface. It's similar to C# StringBuilder class
            Usage as follows :
            <code>
                ErrorString := _stringBuilder
                    .Clear()
                    .Append('Error number: ')
                    .Append(INT_TO_STRING(ErrorNumber))
                    .Append('. Message: ')
                    .Append(ErrorMessage)
                    .Append('.')
                    .ToString();
            </code>

            Inspired by Gerhard Barteling blogpost at https://www.plccoder.com/fluent-code/
    </summary>
</docu>
~*)
FUNCTION_BLOCK StringBuilder
VAR
    {attribute 'hide'}
    _workString : STRING(255);
END_VAR

(*
    Thanks to https://github.com/bengeisler/TcLog
*)
METHOD PROTECTED AnyToString : STRING(255)
VAR_INPUT
    Data : ANY;
END_VAR
VAR
    pAnyBOOL : POINTER TO BOOL;
    pAnyBYTE : POINTER TO BYTE;
    pAnyWORD : POINTER TO WORD;
    pAnyDWORD : POINTER TO DWORD;
    pAnyLWORD : POINTER TO LWORD;
    pAnySINT : POINTER TO SINT;
    pAnyUSINT : POINTER TO USINT;
    pAnyINT : POINTER TO INT;
    pAnyUINT : POINTER TO UINT;
    pAnyDINT : POINTER TO DINT;
    pAnyUDINT : POINTER TO UDINT;
    pAnyLINT : POINTER TO LINT;
    pAnyULINT : POINTER TO ULINT;
    pAnyLTIME : POINTER TO LTIME;
    pAnyReal : POINTER TO REAL;
    pAnyLReal : POINTER TO LREAL;
    pAnyDateAndTime : POINTER TO DATE_AND_TIME;
    pAnyDate : POINTER TO DATE;
    pAnyTime : POINTER TO TIME;
    pAnyWString : POINTER TO WSTRING;
    pAnyTOD : POINTER TO TOD;
    pAnyString : POINTER TO STRING;
    sString : T_MAXSTRING;
    wWString : WSTRING;
END_VAR
IF Data.TypeClass = __SYSTEM.TYPE_CLASS.TYPE_REAL THEN
    pAnyReal := Data.pValue;
    AnyToString := REAL_TO_STRING(pAnyReal^);
ELSIF Data.TypeClass = __SYSTEM.TYPE_CLASS.TYPE_LREAL THEN
    pAnyLReal := Data.pValue;
    AnyToString := LREAL_TO_STRING(pAnyLReal^);
ELSIF Data.TypeClass = __SYSTEM.TYPE_CLASS.TYPE_DATEANDTIME THEN
    pAnyDateAndTime := Data.pValue;
    AnyToString := DT_TO_STRING(pAnyDateAndTime^);
ELSIF Data.TypeClass = __SYSTEM.TYPE_CLASS.TYPE_DATE THEN
    pAnyDate := Data.pValue;
    AnyToString := DATE_TO_STRING(pAnyDate^);
ELSIF Data.TypeClass = __SYSTEM.TYPE_CLASS.TYPE_TIME THEN
    pAnyTime := Data.pValue;
    AnyToString := TIME_TO_STRING(pAnyTime^);
ELSIF Data.TypeClass = __SYSTEM.TYPE_CLASS.TYPE_STRING THEN
    pAnyString := Data.pValue;
    AnyToString := pAnyString^;
ELSIF Data.TypeClass = __SYSTEM.TYPE_CLASS.TYPE_WSTRING THEN
    pAnyWString := Data.pValue;
    wWString := pAnyWString^;
    Tc2_EtherCAT.Tc2_Utilities.WSTRING_TO_STRING2(ADR(sString), ADR(wWstring), SIZEOF(wWString));
    AnyToString := sString;
ELSIF Data.TypeClass = __SYSTEM.TYPE_CLASS.TYPE_TIMEOFDAY THEN
    pAnyTOD := Data.pValue;
    AnyToString := TOD_TO_STRING(pAnyTOD^);
ELSIF Data.TypeClass = __SYSTEM.TYPE_CLASS.TYPE_BOOL THEN
    pAnyBOOL := Data.pValue;
    AnyToString := BOOL_TO_STRING(pAnyBool^);
ELSIF Data.TypeClass = __SYSTEM.TYPE_CLASS.TYPE_BYTE THEN
    pAnyBYTE := Data.pValue;
    AnyToString := BYTE_TO_STRING(pAnyBYTE^);
ELSIF Data.TypeClass = __SYSTEM.TYPE_CLASS.TYPE_WORD THEN
    pAnyWORD := Data.pValue;
    AnyToString := WORD_TO_STRING(pAnyWORD^);
ELSIF Data.TypeClass = __SYSTEM.TYPE_CLASS.TYPE_DWORD THEN
    pAnyDWORD := Data.pValue;
    AnyToString := DWORD_TO_STRING(pAnyDWORD^);
ELSIF Data.TypeClass = __SYSTEM.TYPE_CLASS.TYPE_LWORD THEN
    pAnyLWORD := Data.pValue;
    AnyToString := LWORD_TO_STRING(pAnyLWORD^);
ELSIF Data.TypeClass = __SYSTEM.TYPE_CLASS.TYPE_SINT THEN
    pAnySINT := Data.pValue;
    AnyToString := SINT_TO_STRING(pAnySINT^);
ELSIF Data.TypeClass = __SYSTEM.TYPE_CLASS.TYPE_USINT THEN
    pAnyUSINT := Data.pValue;
    AnyToString := USINT_TO_STRING(pAnyUSINT^);
ELSIF Data.TypeClass = __SYSTEM.TYPE_CLASS.TYPE_INT THEN
    pAnyINT := Data.pValue;
    AnyToString := INT_TO_STRING(pAnyINT^);
ELSIF Data.TypeClass = __SYSTEM.TYPE_CLASS.TYPE_UINT THEN
    pAnyUINT := Data.pValue;
    AnyToString := UINT_TO_STRING(pAnyUINT^);
ELSIF Data.TypeClass = __SYSTEM.TYPE_CLASS.TYPE_DINT THEN
    pAnyDINT := Data.pValue;
    AnyToString := DINT_TO_STRING(pAnyDINT^);
ELSIF Data.TypeClass = __SYSTEM.TYPE_CLASS.TYPE_UDINT THEN
    pAnyUDINT := Data.pValue;
    AnyToString := UDINT_TO_STRING(pAnyUDINT^);
ELSIF Data.TypeClass = __SYSTEM.TYPE_CLASS.TYPE_LINT THEN
    pAnyLINT := Data.pValue;
    AnyToString := LINT_TO_STRING(pAnyLINT^);
ELSIF Data.TypeClass = __SYSTEM.TYPE_CLASS.TYPE_ULINT THEN
    pAnyULINT := Data.pValue;
    AnyToString := ULINT_TO_STRING(pAnyULINT^);
ELSIF Data.TypeClass = __SYSTEM.TYPE_CLASS.TYPE_LTIME THEN
    pAnyLTIME := Data.pValue;
    AnyToString := LTIME_TO_STRING(pAnyLTIME^);
ELSE
    AnyToString := ANY_TO_STRING(Data.pValue^);
END_IF
END_METHOD

METHOD Append : REFERENCE TO StringBuilder
VAR_INPUT
    Text : STRING(255);
END_VAR
_workString := Concat(_workString, text);
Append REF= THIS^;
END_METHOD

METHOD INTERNAL AppendAny : REFERENCE TO StringBuilder
VAR_INPUT
    Data : ANY;
END_VAR
_workString := Concat(_workString, AnyToString(Data));
AppendAny REF= THIS^;
END_METHOD

METHOD Clear : REFERENCE TO StringBuilder
_workString := '';
Clear REF= THIS^;
END_METHOD

METHOD ToString : STRING(255)
ToString := _workString;
END_METHOD

END_FUNCTION_BLOCK

// ---- POUs/Prototypes/TcoLogger/TcoLogger.TcPOU
(*~
        <docu>
            <summary>
                Default implementation of Logger.
                <note type="tip">
                     This type is partially extended by IVF to retrieve messages from the logger in IVF application.
                </note>
            </summary>
            <code>
               // Intializes message retrieval into applications logger
                ..._logger.StartLoggingMessages(eMessageCategory.All);
            </code>
            <code>
                FUNCTION_BLOCK LoggerUsage EXTENDS TcoCore.TcoObject
                VAR
                    _logger : TcoCore.TcoLogger(THIS^);
                    _counter : INT;
                END_VAR
                //---------------------------------------------
                _counter := _counter + 1;
                IF((_counter MOD 100) = 0) THEN
                    _logger.Push('hey friend! we got a problem', eMessageCategory.Critical);
                END_IF;
            </code>
        </docu>
~*)
FUNCTION_BLOCK TcoLogger EXTENDS TcoObject IMPLEMENTS ITcoLogger
VAR
    (*~
        <docu>
            <summary>
                Circural buffer for this logger.
            </summary>
        </docu>
    ~*)
    _buffer : ARRAY[0..MAX_MESSAGE_BUFFER_INDEX] OF TcoLogItem;
    (*~
        <docu>
            <summary>
                Circular carret of of the message buffer.
            </summary>
        </docu>
    ~*)
    _plcCarret : INT;
    (*~
        <docu>
            <summary>
                Minimal log level. Only messages with higher serverity than this will be logged.
            </summary>
        </docu>
    ~*)
    _minLoggingLevel : eMessageCategory := eMessageCategory.Notification;
END_VAR
VAR CONSTANT
    (*~
        <docu>
            <summary>
                Max number of buffered log entries.
            </summary>
        </docu>
    ~*)
    MAX_MESSAGE_BUFFER_INDEX : INT := 1000;
END_VAR

(*~
        <docu>
            <summary>
                Pushes the message to logging buffer.
                See also `PushMessage`
                <note:important>When using this method in a cyclical environment the message will be push each time it is called. You may easily overrun the logging buffer.</note>
            </summary>
        </docu>
~*)
METHOD PUBLIC Push
VAR_INPUT
    (*~
        <docu>
            <summary>
                Message/log entry text.
            </summary>
        </docu>
    ~*)
    Text : STRING(TcoMessengerEnv.MAX_MESSAGE_TEXT_LENGHT);
    (*~
        <docu>
            <summary>
                Message/log entry category.
            </summary>
        </docu>
    ~*)
    Category : eMessageCategory;
END_VAR
VAR
    _tmpMessage : TcoMessage;
END_VAR
IF (Parent <> 0 AND_THEN Parent.Context <> 0 AND_THEN Parent.Context.RealTimeClock <> 0) THEN
    _tmpMessage.TimeStamp := Parent.Context.RealTimeClock.NowLocal();
    _tmpMessage.Cycle := Parent.Context.StartCycleCount;
END_IF;

_tmpMessage.Text := Text;
_tmpMessage.Identity := 0;
_tmpMessage.Category := Category;
_tmpMessage.MessageDigest := 0;
PushMessage(_tmpMessage);
END_METHOD

(*~
        <docu>
            <summary>
                Pushes the message to logging buffer.
                See also `Push`
                <note type="important">
                        This method is typically invoked from a `TcoMessenger`.
                        Depending on settings of the messenger the messages can be logged on rising edge of the message, to prevent buffer overrun.
                        For details see `TcoMessengerSettings`.
                </note>
            </summary>
        </docu>
~*)
METHOD PushMessage
VAR_INPUT
    inMessage : TcoMessage;
END_VAR
IF (inMessage.Category < THIS^._minLoggingLevel OR (THIS^._minLoggingLevel = eMessageCategory.None)) THEN
    RETURN;
END_IF

IF (_plcCarret > MAX_MESSAGE_BUFFER_INDEX) THEN
    _plcCarret := 1;
END_IF

IF (NOT _buffer[_plcCarret].ExpectDequeing) THEN
    _buffer[_plcCarret].Category := inMessage.Category;
    _buffer[_plcCarret].Cycle := inMessage.Cycle;
    _buffer[_plcCarret].ExpectDequeing := TRUE;
    _buffer[_plcCarret].Identity := inMessage.Identity;
    _buffer[_plcCarret].MessageDigest := inMessage.MessageDigest;
    _buffer[_plcCarret].PerCycleCount := inMessage.PerCycleCount;
    _buffer[_plcCarret].Text := inMessage.Text;
    _buffer[_plcCarret].TimeStamp := inMessage.TimeStamp;
    _plcCarret := _plcCarret + 1;
ELSE
    _buffer[0].Text := 'Logging buffer is full we are loosing messages!!!';
    _buffer[0].Category := eMessageCategory.Critical;
    _buffer[0].ExpectDequeing := TRUE;
    _buffer[0].Cycle := THIS^.Context.StartCycleCount;
    _buffer[0].PerCycleCount := _buffer[0].PerCycleCount + 1;
END_IF;
END_METHOD

END_FUNCTION_BLOCK

// ---- POUs/Prototypes/TcoObject/TcoObject.TcPOU
(*~
    <docu>
        <summary>
            Basic construction block from which all blocks of a TcOpen application should derive in order to take advantage of the framework.
            This function block is abstract and must be implemented in a derived block.
            ```TcoObject```, must be constructed via ```FB_init(ITcoObject)``` method at instantiation.
            ```TcoObjects``` that belong to same ```TcoContext``` share the same context.
            This is typically achieved by constructing the object with ```FB_init(THIS^)```, where ```THIS^``` is of ```ITcoObject``` (note that ITcoContext also implements ITcoObject).
            <note type="warning">
                Whenever it is required to pass function block parameters of a block type that derives from `TcoObject` it should be passed as **reference**.
                This means either via appropriate interface or as `REFERENCE TO` in VAR_INPUT and VAR_OUTPUT sections or as VAR_IN_OUT.
                Be aware the VAR_INPUT and VAR_OUTPUT create a copy of the variable.
            </note>
            <para>
                <example>
                <note type="Example">
                <para>
                    All the variables _myContext, _ContextTcoObjectA, _ContextTcoObjectB, _ContextChildTcoObject should have all the same value.
                </para>
                <para>
                    All the variables _myIdentity, _TcoObjectAidentity, _TcoObjectBidentity, _ChildTcoObjectidentity should have uniques values.
                </para>
                    <code>
                            //Definition of the myTcoObject
                            FUNCTION_BLOCK myTcoObject EXTENDS TcoObject
                            VAR
                                  _myChildTcoObject	:	myChildTcoObject(THIS^);
                            END_VAR


                            //Definition of the myTcoContext
                            FUNCTION_BLOCK myTcoContext EXTENDS TcoContext
                            VAR
                                  _myTcoObjectA		:	myTcoObject(THIS^);
                                  _myTcoObjectB		:	myTcoObject(_myTcoObjectA.Context);
                                  _myContext		:	ITcoContext;
                                  _ContextTcoObjectA	:	ITcoContext;
                                  _ContextTcoObjectB	:	ITcoContext;
                                  _ContextChildTcoObject	:	ITcoContext;
                                  _myIdentity		:	ULINT;
                                  _TcoObjectAidentity	: 	ULINT;
                                  _TcoObjectBidentity	: 	ULINT;
                                  _ChildTcoObjectidentity	: 	ULINT;
                            END_VAR

                            //Plc code of the myTcoContext
                            _myContext		:= 		THIS^.Context;
                            _ContextTcoObjectA	:=		_myTcoObjectA.Context;
                            _ContextTcoObjectB	:=		_myTcoObjectB.Context;
                            _ContextChildTcoObject	:=		_myTcoObjectB._myChildTcoObject.Context;
                            _myIdentity		:=		THIS^.Identity;
                            _TcoObjectAidentity	:=		_myTcoObjectA.Identity;
                            _TcoObjectBidentity	:=		_myTcoObjectB.Identity;
                            _ChildTcoObjectidentity	:=		_myTcoObjectB._myChildTcoObject.Identity;
                    </code>
                     <note type="Explanation">
                        <para>
                            The context of the myTcoContext instance is assigned to itself. As the _myTcoObjectA context is assigned to this instance of the myTcoContext, it is assigned to the same context,
                            and the value of the _ContextTcoObjectA will be the same as the value of the _myContext.
                        </para>
                        <para>
                            The context of the _myTcoObjectB instance is assigned to the _myTcoObjectA, that has already assigned context to this instance of the myTcoContext.
                            So the value of the _ContextTcoObjectB will be the same as the values of the _ContextTcoObjectA and _myContext.
                        </para>
                        <para>
                            The context of the _myTcoObjectB._myChildTcoObject instance is assigned to the _myTcoObjectB, that has already assigned context to _myTcoObjectA,
                            that has already assigned its context to this instance of the myTcoContext.
                            So the value of the _ContextChildTcoObject wile be the same as the values _ContextTcoObjectB,_ContextTcoObjectA and _myContext.
                        </para>
                        <para>
                            As the Identities of all objects points to the themselves, all identities will have different values, as all objects are unique.
                        </para>
                     </note>
                 </note>
                </example>
            </para>
         </summary>
    </docu>
~*)
{attribute addProperty ToolTip ""}
{attribute 'no_assign'}
FUNCTION_BLOCK ABSTRACT TcoObject IMPLEMENTS ITcoObject
VAR
    {attribute clr [RenderIgnore()]}
    {attribute clr [ReadOnly()]}
    {attribute clr [CompilerOmits("BuilderPlainer", "BuilderShadow")]}
    _Identity : ULINT;
    {attribute 'hide'}
    _ParentObject : ITcoObject;
    {attribute 'hide'}
    _ParentStruct : REFERENCE TO TcoStruct;
    {attribute clr [RenderIgnore()]}
    {attribute clr [CompilerOmits("BuilderPlainer", "BuilderShadow")]}
    _messenger : TcoMessenger(THIS^);
END_VAR

(*~
    <docu>
        <summary>
            Gets the context of the this object. The context is provided by parent object(s).
        </summary>
    </docu>
~*)
PROPERTY PUBLIC Context : ITcoContext
GET
Context := THIS^.Parent.Context;
END_GET
END_PROPERTY

(*~
    <docu>
        <summary>
            Compares this object to another object and returns ```true``` when the reference equals.
            When overriden in derived class custom comparison of two objects of the same type can be evaluated.
         </summary>
        <note>
            Default implementation compares only if two objects share the same reference.
            If you want to compare actual values of the objects you will need to override EqualsTo method,
            where you evaluate the values for equality.
        </note>
        <example>
            <code>
                // EqualsTo method override example of type MyObject
                METHOD PUBLIC EqualsTo : BOOL
                VAR_INPUT
                    Object : ITcoObject;
                END_VAR

                VAR
                    _object : POINTER TO MyObject;
                END_VAR
                //--------------------------------------------
                IF(__QUERYPOINTER(Object,  _object)) THEN
                    EqualsTo := _object^._SomeNumber = THIS^._SomeNumber AND _object^._SomeString = THIS^._SomeString;
                END_IF;
            </code>
        </example>
    </docu>
~*)
METHOD PUBLIC EqualsTo : BOOL
VAR_INPUT
    Object : ITcoObject;
END_VAR
IF (Object.Identity <> 0) THEN
    EqualsTo := Object.Identity = THIS^.Identity;
END_IF
END_METHOD

{attribute 'hide'}
METHOD FB_init : BOOL
VAR_INPUT
    bInitRetains : BOOL; // if TRUE, the retain variables are initialized (warm start / cold start)
    bInCopyCode : BOOL; // if TRUE, the instance afterwards gets moved into the copy code (online change)
    ParentObject : ITcoObject;
END_VAR
_Identity := ADR(THIS^);
_ParentObject := ParentObject;
END_METHOD

(*~
    <docu>
        <summary>
            Gets the identity of this <see cref ="PlcDocu.TcoCore.TcoObject()"/>.
            This value is assigned after download by calling the implicit method <c>FB_init()</c> and cannot be changed during runtime.
            This variable is used in the higher level applications.
        </summary>
    </docu>
~*)
PROPERTY Identity : ULINT
GET
_Identity := ADR(THIS^);
Identity := _Identity;
END_GET
END_PROPERTY

(*~
        <docu>
            <summary>
                Gets messenger of this object.
                See <see cref="PlcDocu.TcoCore.TcoMessenger()"/> for more details.
            </summary>
        </docu>
~*)
PROPERTY Messenger : ITcoMessenger
GET
Messenger := THIS^._messenger;
END_GET
END_PROPERTY

PROPERTY Parent : ITcoObject
GET
IF (_ParentObject <> 0) THEN
    Parent := _ParentObject;
    RETURN;
END_IF;

IF (__ISVALIDREF(_ParentStruct) AND_THEN _ParentStruct.Parent <> 0) THEN
    Parent := _ParentStruct.Parent;
    RETURN;
END_IF;
END_GET
END_PROPERTY

END_FUNCTION_BLOCK

// ---- POUs/Prototypes/TcoMessage/TcoMessenger.TcPOU
(*~
        <docu>
            <summary>
                Provides mechanism for delivering static messages to the supervising applications (SCADA/HMI).
                <remarks>
                    <note type="important">
                        Each messenger has a single placeholder for the message; it stores the most important message from the last context cycle.
                        If there are more messages in a single cycle for the same messenger then less important messages are discarded and replaced by
                        the message with the category of higher severity.
                    </note>
                    <note type="important">
                        Messenger can send the data to context logger. There is a maximum limit of 10 different messages per messenger in 2 consecutive context cycles.
                        The messages that exceed this limit won't be logged when `OnEventRisen` logging is set.
                        Take this behaviour into account when designing your system.
                    </note>
                </remarks>
            </summary>

        </docu>
~*)
FUNCTION_BLOCK PUBLIC TcoMessenger IMPLEMENTS ITcoMessenger, ITcoMessageProperties, ITcoMessageTextBuilder, ITcoMessageCategorize
VAR
    (*~
        <docu>
            <summary>
                Most important message of this instance of messenger; stores the most important message from the last context cycle.
                If there are more messages in a single cycle for the same
                messenger then less important messages are discarded and replaced by the message with the category of higher severity.
            </summary>
        </docu>
    ~*)
    _mime : TcoMessage;
    _Parent : ITcoObject;
    {attribute clr [ReadOnly()]}
    _contextIdentity : ULINT;
    {attribute 'hide'}
    _mds : ARRAY[0..MDS_MAX_INDEX] OF TcoMessageDigest;
    {attribute 'hide'}
    _condition : eMessageCondition;
    {attribute 'hide'}
    _pinnable : BOOL;
END_VAR
VAR
    {attribute 'hide'}
    tmpMessageText : STRING(TcoMessengerEnv.MAX_MESSAGE_TEXT_LENGHT);
    {attribute 'hide'}
    refStringBuilder : REFERENCE TO StringBuilder;
END_VAR
VAR CONSTANT
    MDS_MAX_INDEX : INT := 10;
END_VAR
VAR_STAT
    {attribute 'hide'}
    _conflictingStringBuilder : StringBuilder;
END_VAR

(*~
    <docu>
        <summary>
            Appends string to the message text.
        </summary>
        <remarks>
            <note type="warning">
                The size of the resulting string should not be more than '160' characters. The characters exceeding this size will be truncated.
            </note>
        </remarks>
    </docu>
~*)
{attribute 'hide'}
{attribute 'obsolete' := 'This method must be accessed ITcoMessageTextBuilder interface'}
METHOD Append : ITcoMessageTextBuilder
VAR_INPUT
    Text : STRING(TcoMessengerEnv.MAX_MESSAGE_TEXT_LENGHT);
END_VAR
THIS^.StringBuilder.Append(Text);
Append := THIS^;
END_METHOD

(*~
    <docu>
        <summary>
            Appends any value to the message text.
        </summary>
        <remarks>
            <note type="warning">
                The size of the resulting string should not be more than '160' characters. The characters exceeding this size will be truncated.
            </note>
        </remarks>
    </docu>
~*)
METHOD AppendAny : ITcoMessageTextBuilder
VAR_INPUT
    Data : ANY;
END_VAR
THIS^.StringBuilder.AppendAny(Data);
AppendAny := THIS^;
END_METHOD

(*~
    <docu>
        <summary>
            Gets categorization methods for fluent message builder.
        </summary>
    </docu>
~*)
{attribute 'hide'}
{attribute 'obsolete' := 'This method must be accessed ITcoMessageTextBuilder interface'}
METHOD As : ITcoMessageCategorize
As := THIS^;
END_METHOD

(*~
        <docu>
            <summary>
                Categotizes and creates the message as  'debug'.
            </summary>
        </docu>
~*)
{attribute 'hide'}
{attribute 'obsolete' := 'This method must be accessed ITcoMessageCategorize interface'}
METHOD PUBLIC AsDebug : ITcoMessageProperties
AsDebug := Post(THIS^.StringBuilder.ToString(), eMessageCategory.Debug);
END_METHOD

(*~
        <docu>
            <summary>
                Categotizes and creates the message as  'error'.
            </summary>
        </docu>
~*)
{attribute 'hide'}
{attribute 'obsolete' := 'This method must be accessed ITcoMessageCategorize interface'}
METHOD PUBLIC AsError : ITcoMessageProperties
AsError := Post(THIS^.StringBuilder.ToString(), eMessageCategory.Error);
END_METHOD

(*~
        <docu>
            <summary>
                Categotizes and creates the message as  'fatal'.
            </summary>
        </docu>
~*)
{attribute 'hide'}
{attribute 'obsolete' := 'This method must be accessed ITcoMessageCategorize interface'}
METHOD PUBLIC AsFatal : ITcoMessageProperties
AsFatal := Post(THIS^.StringBuilder.ToString(), eMessageCategory.Fatal);
END_METHOD

(*~
        <docu>
            <summary>
                Categotizes and creates the message as  'information'.
            </summary>
        </docu>
~*)
{attribute 'hide'}
{attribute 'obsolete' := 'This method must be accessed ITcoMessageCategorize interface'}
METHOD PUBLIC AsInfo : ITcoMessageProperties
AsInfo := Post(THIS^.StringBuilder.ToString(), eMessageCategory.Info);
END_METHOD

(*~
        <docu>
            <summary>
                Categotizes and creates the message as  'trace'.
            </summary>
        </docu>
~*)
{attribute 'hide'}
{attribute 'obsolete' := 'This method must be accessed ITcoMessageCategorize interface'}
METHOD PUBLIC AsTrace : ITcoMessageProperties
AsTrace := Post(THIS^.StringBuilder.ToString(), eMessageCategory.Trace);
END_METHOD

(*~
        <docu>
            <summary>
                Categotizes and creates the message as 'warning'.
            </summary>
        </docu>
~*)
{attribute 'hide'}
{attribute 'obsolete' := 'This method must be accessed ITcoMessageCategorize interface'}
METHOD PUBLIC AsWarning : ITcoMessageProperties
AsWarning := Post(THIS^.StringBuilder.ToString(), eMessageCategory.Warning);
END_METHOD

(*~
    <docu>
        <summary>
            Initiates new message text building for this messenger in fluent-like fashion.
        </summary>
    </docu>
~*)
METHOD Build : ITcoMessageTextBuilder
THIS^.StringBuilder.Clear();
Build := THIS^;
END_METHOD

(*~
        <docu>
            <summary>
                Adds message of 'catastrophic' category to the message queue.
                Use this category when there is a situation when the device cannot continue operations due to irrecoverable failure.
            </summary>
        </docu>
~*)
METHOD PUBLIC Catastrophic : ITcoMessageProperties
VAR_INPUT
    (*~
        <docu>
            <summary>
                Arbitrary message string.
            </summary>
        </docu>
    ~*)
    Message : STRING(TcoMessengerEnv.MAX_MESSAGE_TEXT_LENGHT);
END_VAR
Catastrophic := THIS^.Post(Message, eMessageCategory.Catastrophic);
END_METHOD

